LIN {X 0,Y 145.306,Z 169.772,A -85,B 0,C 180,E1 -24522.343,E2 -24522.343} C_VEL
LIN {X 0,Y 146.509,Z 171.03,A -85,B 0,C 180,E1 -24522.943,E2 -24522.943} C_VEL
LIN {X 0,Y 148.712,Z 174.406,A -85,B 0,C 180,E1 -24524.074,E2 -24524.074} C_VEL
LIN {X 0,Y 152.72,Z 180.292,A -85,B 0,C 180,E1 -24525.978,E2 -24525.978} C_VEL
LIN {X 0,Y 157.75,Z 189.892,A -85,B 0,C 180,E1 -24528.287,E2 -24528.287} C_VEL
LIN {X 0,Y 163.669,Z 203.505,A -85,B 0,C 180,E1 -24530.86,E2 -24530.86} C_VEL
LIN {X 0,Y 165.632,Z 209.272,A -85,B 0,C 180,E1 -24531.721,E2 -24531.721} C_VEL
LIN {X 0,Y 166.47,Z 218.611,A -85,B 0,C 180,E1 -24532.446,E2 -24532.446} C_VEL
LIN {X 0,Y 165.086,Z 241.604,A -85,B 0,C 180,E1 -24533.417,E2 -24533.417} C_VEL
LIN {X 0,Y 163.759,Z 252.442,A -85,B 0,C 180,E1 -24534.195,E2 -24534.195} C_VEL
LIN {X 0,Y 161.522,Z 264.21,A -85,B 0,C 180,E1 -24535.554,E2 -24535.554} C_VEL
LIN {X 0,Y 159.643,Z 271.971,A -85,B 0,C 180,E1 -24536.766,E2 -24536.766} C_VEL
LIN {X 0,Y 157.428,Z 279.918,A -85,B 0,C 180,E1 -24538.363,E2 -24538.363} C_VEL
LIN {X 0,Y 154.747,Z 287.967,A -85,B 0,C 180,E1 -24540.404,E2 -24540.404} C_VEL
LIN {X 0,Y 152.242,Z 294.615,A -85,B 0,C 180,E1 -24542.508,E2 -24542.508} C_VEL
LIN {X 0,Y 149.733,Z 300.93,A -85,B 0,C 180,E1 -24545.013,E2 -24545.013} C_VEL
LIN {X 0,Y 147.469,Z 306.176,A -85,B 0,C 180,E1 -24547.589,E2 -24547.589} C_VEL
LIN {X 0,Y 145.528,Z 310.551,A -85,B 0,C 180,E1 -24550.243,E2 -24550.243} C_VEL
LIN {X 0,Y 143.291,Z 315.716,A -85,B 0,C 180,E1 -24554.351,E2 -24554.351} C_VEL
LIN {X 0,Y 141.729,Z 319.509,A -85,B 0,C 180,E1 -24558.56,E2 -24558.56} C_VEL
LIN {X 0,Y 141.028,Z 321.248,A -85,B 0,C 180,E1 -24561.403,E2 -24561.403} C_VEL
LIN {X 0,Y 140.636,Z 322.494,A -85,B 0,C 180,E1 -24564.265,E2 -24564.265} C_VEL
LIN {X 0,Y 140.489,Z 323.267,A -85,B 0,C 180,E1 -24567.133,E2 -24567.133} C_VEL
LIN {X 0,Y 140.527,Z 323.559,A -85,B 0,C 180,E1 -24570.001,E2 -24570.001} C_VEL
LIN {X 0,Y 140.489,Z 323.255,A -85,B 0,C 180,E1 -24572.868,E2 -24572.868} C_VEL
LIN {X 0,Y 140.635,Z 322.459,A -85,B 0,C 180,E1 -24575.737,E2 -24575.737} C_VEL
LIN {X 0,Y 141.018,Z 321.189,A -85,B 0,C 180,E1 -24578.599,E2 -24578.599} C_VEL
LIN {X 0,Y 142.198,Z 318.101,A -85,B 0,C 180,E1 -24583.058,E2 -24583.058} C_VEL
LIN {X 0,Y 143.967,Z 314.085,A -85,B 0,C 180,E1 -24587.032,E2 -24587.032} C_VEL
LIN {X 0,Y 146.467,Z 308.354,A -85,B 0,C 180,E1 -24591.093,E2 -24591.093} C_VEL
LIN {X 0,Y 148.407,Z 303.949,A -85,B 0,C 180,E1 -24593.51,E2 -24593.51} C_VEL
LIN {X 0,Y 149.365,Z 300.401,A -85,B 0,C 180,E1 -24595.293,E2 -24595.293} C_VEL
LIN {X 0,Y 149.331,Z 294.144,A -85,B 0,C 180,E1 -24598.252,E2 -24598.252} C_VEL
LIN {X 0,Y 149.369,Z 287.186,A -85,B 0,C 180,E1 -24600.965,E2 -24600.965} C_VEL
LIN {X 0,Y 150.382,Z 282.536,A -85,B 0,C 180,E1 -24602.304,E2 -24602.304} C_VEL
LIN {X 0,Y 152.699,Z 275.158,A -85,B 0,C 180,E1 -24603.961,E2 -24603.961} C_VEL
LIN {X 0,Y 154.808,Z 267.286,A -85,B 0,C 180,E1 -24605.368,E2 -24605.368} C_VEL
LIN {X 0,Y 156.648,Z 258.957,A -85,B 0,C 180,E1 -24606.521,E2 -24606.521} C_VEL
LIN {X 0,Y 158.362,Z 249.266,A -85,B 0,C 180,E1 -24607.478,E2 -24607.478} C_VEL
LIN {X 0,Y 159.434,Z 239.95,A -85,B 0,C 180,E1 -24608.108,E2 -24608.108} C_VEL
LIN {X 0,Y 160.713,Z 217.708,A -85,B 0,C 180,E1 -24609.076,E2 -24609.076} C_VEL
LIN {X 0,Y 159.799,Z 210.505,A -85,B 0,C 180,E1 -24609.751,E2 -24609.751} C_VEL
LIN {X 0,Y 156.697,Z 202.354,A -85,B 0,C 180,E1 -24611.18,E2 -24611.18} C_VEL
LIN {X 0,Y 151.188,Z 189.975,A -85,B 0,C 180,E1 -24613.813,E2 -24613.813} C_VEL
LIN {X 0,Y 147.611,Z 183.574,A -85,B 0,C 180,E1 -24615.587,E2 -24615.587} C_VEL
LIN {X 0,Y 144.362,Z 178.907,A -85,B 0,C 180,E1 -24617.245,E2 -24617.245} C_VEL
LIN {X 0,Y 142.077,Z 175.537,A -85,B 0,C 180,E1 -24618.496,E2 -24618.496} C_VEL
LIN {X 0,Y 139.925,Z 172.519,A -85,B 0,C 180,E1 -24619.73,E2 -24619.73} C_VEL
LIN {X 0,Y 139.2,Z 171.415,A -85,B 0,C 180,E1 -24620.169,E2 -24620.169} C_VEL
LIN {X 0,Y 137.076,Z 169.279,A -85,B 0,C 180,E1 -24621.414,E2 -24621.414} C_VEL
LIN {X 0,Y 136.185,Z 167.112,A -85,B 0,C 180,E1 -24622.206,E2 -24622.206} C_VEL
LIN {X 0,Y 136.03,Z 166.393,A -85,B 0,C 180,E1 -24623.087,E2 -24623.087} C_VEL
LIN {X 0,Y 136.086,Z 166.344,A -85,B 0,C 180,E1 -24628.907,E2 -24628.907} C_VEL
LIN {X 0,Y 136.149,Z 166.308,A -85,B 0,C 180,E1 -24632.317,E2 -24632.317} C_VEL
LIN {X 0,Y 136.246,Z 166.297,A -85,B 0,C 180,E1 -24638.834,E2 -24638.834} C_VEL
LIN {X 0,Y 136.278,Z 166.322,A -85,B 0,C 180,E1 -24645.058,E2 -24645.058} C_VEL
LIN {X 0,Y 136.447,Z 166.265,A -85,B 0,C 180,E1 -24648.138,E2 -24648.138} C_VEL
LIN {X 0,Y 136.555,Z 166.253,A -85,B 0,C 180,E1 -24651.118,E2 -24651.118} C_VEL
LIN {X 0,Y 137.135,Z 166.174,A -85,B 0,C 180,E1 -24660,E2 -24660} C_VEL
LIN {X 0,Y 136.582,Z 166.243,A -85,B 0,C 180,E1 -24668.881,E2 -24668.881} C_VEL
LIN {X 0,Y 136.494,Z 166.277,A -85,B 0,C 180,E1 -24671.955,E2 -24671.955} C_VEL
LIN {X 0,Y 136.254,Z 166.287,A -85,B 0,C 180,E1 -24678.028,E2 -24678.028} C_VEL
LIN {X 0,Y 136.205,Z 166.325,A -85,B 0,C 180,E1 -24681.754,E2 -24681.754} C_VEL
LIN {X 0,Y 136.121,Z 166.321,A -85,B 0,C 180,E1 -24688.63,E2 -24688.63} C_VEL
LIN {X 0,Y 136.046,Z 166.327,A -85,B 0,C 180,E1 -24694.629,E2 -24694.629} C_VEL
LIN {X 0,Y 136.087,Z 166.637,A -85,B 0,C 180,E1 -24697.709,E2 -24697.709} C_VEL
LIN {X 0,Y 136.369,Z 167.781,A -85,B 0,C 180,E1 -24698.358,E2 -24698.358} C_VEL
LIN {X 0,Y 137.896,Z 170.333,A -85,B 0,C 180,E1 -24699.393,E2 -24699.393} C_VEL
LIN {X 0,Y 139.623,Z 171.907,A -85,B 0,C 180,E1 -24700.376,E2 -24700.376} C_VEL
LIN {X 0,Y 141.835,Z 175.359,A -85,B 0,C 180,E1 -24701.68,E2 -24701.68} C_VEL
LIN {X 0,Y 143.196,Z 177.113,A -85,B 0,C 180,E1 -24702.42,E2 -24702.42} C_VEL
LIN {X 0,Y 148.232,Z 184.462,A -85,B 0,C 180,E1 -24705.016,E2 -24705.016} C_VEL
LIN {X 0,Y 154.436,Z 194.858,A -85,B 0,C 180,E1 -24707.927,E2 -24707.927} C_VEL
LIN {X 0,Y 158.358,Z 202.506,A -85,B 0,C 180,E1 -24709.65,E2 -24709.65} C_VEL
LIN {X 0,Y 161.183,Z 209.91,A -85,B 0,C 180,E1 -24710.921,E2 -24710.921} C_VEL
LIN {X 0,Y 159.528,Z 236.911,A -85,B 0,C 180,E1 -24712.08,E2 -24712.08} C_VEL
LIN {X 0,Y 158.138,Z 248.435,A -85,B 0,C 180,E1 -24712.962,E2 -24712.962} C_VEL
LIN {X 0,Y 156.015,Z 259.714,A -85,B 0,C 180,E1 -24714.358,E2 -24714.358} C_VEL
LIN {X 0,Y 153.691,Z 269.059,A -85,B 0,C 180,E1 -24715.937,E2 -24715.937} C_VEL
LIN {X 0,Y 151.299,Z 277.142,A -85,B 0,C 180,E1 -24717.711,E2 -24717.711} C_VEL
LIN {X 0,Y 148.543,Z 284.842,A -85,B 0,C 180,E1 -24719.821,E2 -24719.821} C_VEL
LIN {X 0,Y 145.37,Z 292.896,A -85,B 0,C 180,E1 -24722.658,E2 -24722.658} C_VEL
LIN {X 0,Y 142.292,Z 299.943,A -85,B 0,C 180,E1 -24725.953,E2 -24725.953} C_VEL
LIN {X 0,Y 139.612,Z 305.513,A -85,B 0,C 180,E1 -24729.367,E2 -24729.367} C_VEL
LIN {X 0,Y 137.099,Z 310.686,A -85,B 0,C 180,E1 -24733.623,E2 -24733.623} C_VEL
LIN {X 0,Y 135.79,Z 313.338,A -85,B 0,C 180,E1 -24736.531,E2 -24736.531} C_VEL
LIN {X 0,Y 134.441,Z 316.24,A -85,B 0,C 180,E1 -24740.976,E2 -24740.976} C_VEL
LIN {X 0,Y 133.881,Z 317.504,A -85,B 0,C 180,E1 -24743.973,E2 -24743.973} C_VEL
LIN {X 0,Y 133.534,Z 318.299,A -85,B 0,C 180,E1 -24746.982,E2 -24746.982} C_VEL
LIN {X 0,Y 133.475,Z 318.601,A -85,B 0,C 180,E1 -24749.999,E2 -24749.999} C_VEL
LIN {X 0,Y 133.534,Z 318.32,A -85,B 0,C 180,E1 -24753.016,E2 -24753.016} C_VEL
LIN {X 0,Y 133.877,Z 317.568,A -85,B 0,C 180,E1 -24756.026,E2 -24756.026} C_VEL
LIN {X 0,Y 134.371,Z 316.349,A -85,B 0,C 180,E1 -24759.027,E2 -24759.027} C_VEL
LIN {X 0,Y 135.782,Z 313.49,A -85,B 0,C 180,E1 -24763.468,E2 -24763.468} C_VEL
LIN {X 0,Y 137.051,Z 310.887,A -85,B 0,C 180,E1 -24766.381,E2 -24766.381} C_VEL
LIN {X 0,Y 139.57,Z 305.767,A -85,B 0,C 180,E1 -24770.638,E2 -24770.638} C_VEL
LIN {X 0,Y 142.234,Z 300.257,A -85,B 0,C 180,E1 -24774.056,E2 -24774.056} C_VEL
LIN {X 0,Y 145.279,Z 293.329,A -85,B 0,C 180,E1 -24777.359,E2 -24777.359} C_VEL
LIN {X 0,Y 148.49,Z 285.371,A -85,B 0,C 180,E1 -24780.19,E2 -24780.19} C_VEL
LIN {X 0,Y 151.263,Z 277.782,A -85,B 0,C 180,E1 -24782.296,E2 -24782.296} C_VEL
LIN {X 0,Y 153.628,Z 269.829,A -85,B 0,C 180,E1 -24784.082,E2 -24784.082} C_VEL
LIN {X 0,Y 155.656,Z 262.251,A -85,B 0,C 180,E1 -24785.403,E2 -24785.403} C_VEL
LIN {X 0,Y 157.548,Z 252.986,A -85,B 0,C 180,E1 -24786.671,E2 -24786.671} C_VEL
LIN {X 0,Y 158.99,Z 243.674,A -85,B 0,C 180,E1 -24787.591,E2 -24787.591} C_VEL
LIN {X 0,Y 159.965,Z 233.274,A -85,B 0,C 180,E1 -24788.286,E2 -24788.286} C_VEL
LIN {X 0,Y 161.313,Z 209.971,A -85,B 0,C 180,E1 -24789.247,E2 -24789.247} C_VEL
LIN {X 0,Y 157.275,Z 199.981,A -85,B 0,C 180,E1 -24791.055,E2 -24791.055} C_VEL
LIN {X 0,Y 151.741,Z 190.114,A -85,B 0,C 180,E1 -24793.537,E2 -24793.537} C_VEL
LIN {X 0,Y 145.574,Z 180.386,A -85,B 0,C 180,E1 -24796.579,E2 -24796.579} C_VEL
LIN {X 0,Y 142.966,Z 176.681,A -85,B 0,C 180,E1 -24797.972,E2 -24797.972} C_VEL
LIN {X 0,Y 139.995,Z 172.674,A -85,B 0,C 180,E1 -24799.655,E2 -24799.655} C_VEL
LIN {X 0,Y 139.171,Z 171.41,A -85,B 0,C 180,E1 -24800.157,E2 -24800.157} C_VEL
LIN {X 0,Y 136.985,Z 169.121,A -85,B 0,C 180,E1 -24801.459,E2 -24801.459} C_VEL
LIN {X 0,Y 136.181,Z 167.095,A -85,B 0,C 180,E1 -24802.204,E2 -24802.204} C_VEL
LIN {X 0,Y 136.027,Z 166.389,A -85,B 0,C 180,E1 -24803.085,E2 -24803.085} C_VEL
LIN {X 0,Y 136.066,Z 166.34,A -85,B 0,C 180,E1 -24808.901,E2 -24808.901} C_VEL
LIN {X 0,Y 136.147,Z 166.311,A -85,B 0,C 180,E1 -24812.316,E2 -24812.316} C_VEL
LIN {X 0,Y 136.247,Z 166.312,A -85,B 0,C 180,E1 -24818.833,E2 -24818.833} C_VEL
LIN {X 0,Y 136.283,Z 166.31,A -85,B 0,C 180,E1 -24825.057,E2 -24825.057} C_VEL
LIN {X 0,Y 136.496,Z 166.277,A -85,B 0,C 180,E1 -24828.114,E2 -24828.114} C_VEL
LIN {X 0,Y 136.578,Z 166.243,A -85,B 0,C 180,E1 -24831.119,E2 -24831.119} C_VEL
LIN {X 0,Y 137.133,Z 166.175,A -85,B 0,C 180,E1 -24840,E2 -24840} C_VEL
LIN {X 0,Y 136.591,Z 166.249,A -85,B 0,C 180,E1 -24848.879,E2 -24848.879} C_VEL
LIN {X 0,Y 136.49,Z 166.261,A -85,B 0,C 180,E1 -24851.954,E2 -24851.954} C_VEL
LIN {X 0,Y 136.251,Z 166.296,A -85,B 0,C 180,E1 -24858.028,E2 -24858.028} C_VEL
LIN {X 0,Y 136.197,Z 166.309,A -85,B 0,C 180,E1 -24861.749,E2 -24861.749} C_VEL
LIN {X 0,Y 136.117,Z 166.314,A -85,B 0,C 180,E1 -24868.63,E2 -24868.63} C_VEL
LIN {X 0,Y 136.043,Z 166.328,A -85,B 0,C 180,E1 -24874.629,E2 -24874.629} C_VEL
LIN {X 0,Y 136.07,Z 166.645,A -85,B 0,C 180,E1 -24877.19,E2 -24877.19} C_VEL
LIN {X 0,Y 136.364,Z 167.734,A -85,B 0,C 180,E1 -24877.852,E2 -24877.852} C_VEL
LIN {X 0,Y 137.89,Z 170.334,A -85,B 0,C 180,E1 -24878.902,E2 -24878.902} C_VEL
LIN {X 0,Y 139.615,Z 171.833,A -85,B 0,C 180,E1 -24879.885,E2 -24879.885} C_VEL
LIN {X 0,Y 141.706,Z 175.185,A -85,B 0,C 180,E1 -24881.136,E2 -24881.136} C_VEL
LIN {X 0,Y 143.181,Z 177.043,A -85,B 0,C 180,E1 -24881.941,E2 -24881.941} C_VEL
LIN {X 0,Y 148.421,Z 184.735,A -85,B 0,C 180,E1 -24884.658,E2 -24884.658} C_VEL
LIN {X 0,Y 153.079,Z 193.843,A -85,B 0,C 180,E1 -24886.964,E2 -24886.964} C_VEL
LIN {X 0,Y 159.051,Z 207.999,A -85,B 0,C 180,E1 -24889.758,E2 -24889.758} C_VEL
LIN {X 0,Y 160.238,Z 211.76,A -85,B 0,C 180,E1 -24890.33,E2 -24890.33} C_VEL
LIN {X 0,Y 160.859,Z 219.504,A -85,B 0,C 180,E1 -24890.949,E2 -24890.949} C_VEL
LIN {X 0,Y 159.439,Z 241.491,A -85,B 0,C 180,E1 -24891.895,E2 -24891.895} C_VEL
LIN {X 0,Y 157.96,Z 253.007,A -85,B 0,C 180,E1 -24892.753,E2 -24892.753} C_VEL
LIN {X 0,Y 155.717,Z 264.088,A -85,B 0,C 180,E1 -24894.075,E2 -24894.075} C_VEL
LIN {X 0,Y 153.481,Z 272.848,A -85,B 0,C 180,E1 -24895.51,E2 -24895.51} C_VEL
LIN {X 0,Y 151.018,Z 281.024,A -85,B 0,C 180,E1 -24897.249,E2 -24897.249} C_VEL
LIN {X 0,Y 148.226,Z 288.863,A -85,B 0,C 180,E1 -24899.357,E2 -24899.357} C_VEL
LIN {X 0,Y 145.323,Z 296.197,A -85,B 0,C 180,E1 -24901.868,E2 -24901.868} C_VEL
LIN {X 0,Y 142.115,Z 303.636,A -85,B 0,C 180,E1 -24905.144,E2 -24905.144} C_VEL
LIN {X 0,Y 139.371,Z 309.466,A -85,B 0,C 180,E1 -24908.557,E2 -24908.557} C_VEL
LIN {X 0,Y 137.189,Z 314.066,A -85,B 0,C 180,E1 -24912.1,E2 -24912.1} C_VEL
LIN {X 0,Y 135.811,Z 317.057,A -85,B 0,C 180,E1 -24915.005,E2 -24915.005} C_VEL
LIN {X 0,Y 134.77,Z 319.381,A -85,B 0,C 180,E1 -24917.961,E2 -24917.961} C_VEL
LIN {X 0,Y 134.003,Z 321.12,A -85,B 0,C 180,E1 -24920.948,E2 -24920.948} C_VEL
LIN {X 0,Y 133.566,Z 322.365,A -85,B 0,C 180,E1 -24923.96,E2 -24923.96} C_VEL
LIN {X 0,Y 133.401,Z 323.138,A -85,B 0,C 180,E1 -24926.981,E2 -24926.981} C_VEL
LIN {X 0,Y 133.448,Z 323.431,A -85,B 0,C 180,E1 -24930.001,E2 -24930.001} C_VEL
LIN {X 0,Y 133.401,Z 323.126,A -85,B 0,C 180,E1 -24933.021,E2 -24933.021} C_VEL
LIN {X 0,Y 133.565,Z 322.33,A -85,B 0,C 180,E1 -24936.042,E2 -24936.042} C_VEL
LIN {X 0,Y 133.992,Z 321.06,A -85,B 0,C 180,E1 -24939.054,E2 -24939.054} C_VEL
LIN {X 0,Y 135.202,Z 318.139,A -85,B 0,C 180,E1 -24943.528,E2 -24943.528} C_VEL
LIN {X 0,Y 136.426,Z 315.477,A -85,B 0,C 180,E1 -24946.46,E2 -24946.46} C_VEL
LIN {X 0,Y 138.841,Z 310.281,A -85,B 0,C 180,E1 -24950.753,E2 -24950.753} C_VEL
LIN {X 0,Y 142.111,Z 303.43,A -85,B 0,C 180,E1 -24954.858,E2 -24954.858} C_VEL
LIN {X 0,Y 145.329,Z 295.948,A -85,B 0,C 180,E1 -24958.133,E2 -24958.133} C_VEL
LIN {X 0,Y 148.195,Z 288.568,A -85,B 0,C 180,E1 -24960.652,E2 -24960.652} C_VEL
LIN {X 0,Y 150.382,Z 282.536,A -85,B 0,C 180,E1 -24962.304,E2 -24962.304} C_VEL
LIN {X 0,Y 151.374,Z 277.866,A -85,B 0,C 180,E1 -24963.554,E2 -24963.554} C_VEL
LIN {X 0,Y 151.28,Z 269.925,A -85,B 0,C 180,E1 -24965.711,E2 -24965.711} C_VEL
LIN {X 0,Y 151.137,Z 261.247,A -85,B 0,C 180,E1 -24967.658,E2 -24967.658} C_VEL
LIN {X 0,Y 151.671,Z 255.69,A -85,B 0,C 180,E1 -24968.473,E2 -24968.473} C_VEL
LIN {X 0,Y 153.583,Z 243.837,A -85,B 0,C 180,E1 -24969.505,E2 -24969.505} C_VEL
LIN {X 0,Y 154.8,Z 226.982,A -85,B 0,C 180,E1 -24970.312,E2 -24970.312} C_VEL
LIN {X 0,Y 155.171,Z 218.327,A -85,B 0,C 180,E1 -24970.711,E2 -24970.711} C_VEL
LIN {X 0,Y 154.459,Z 212.838,A -85,B 0,C 180,E1 -24971.269,E2 -24971.269} C_VEL
LIN {X 0,Y 149.342,Z 199.941,A -85,B 0,C 180,E1 -24973.84,E2 -24973.84} C_VEL
LIN {X 0,Y 144.771,Z 190.32,A -85,B 0,C 180,E1 -24976.265,E2 -24976.265} C_VEL
LIN {X 0,Y 140.402,Z 183.75,A -85,B 0,C 180,E1 -24978.646,E2 -24978.646} C_VEL
LIN {X 0,Y 138.218,Z 180.588,A -85,B 0,C 180,E1 -24979.928,E2 -24979.928} C_VEL
LIN {X 0,Y 135.858,Z 177.165,A -85,B 0,C 180,E1 -24981.402,E2 -24981.402} C_VEL
LIN {X 0,Y 133.57,Z 174.376,A -85,B 0,C 180,E1 -24982.883,E2 -24982.883} C_VEL
LIN {X 0,Y 132.566,Z 172.525,A -85,B 0,C 180,E1 -24983.623,E2 -24983.623} C_VEL
LIN {X 0,Y 130.346,Z 170.554,A -85,B 0,C 180,E1 -24985.146,E2 -24985.146} C_VEL
LIN {X 0,Y 129.15,Z 167.989,A -85,B 0,C 180,E1 -24986.323,E2 -24986.323} C_VEL
LIN {X 0,Y 129.005,Z 167.269,A -85,B 0,C 180,E1 -24987.455,E2 -24987.455} C_VEL
LIN {X 0,Y 129.052,Z 167.197,A -85,B 0,C 180,E1 -24990.652,E2 -24990.652} C_VEL
LIN {X 0,Y 129.109,Z 167.195,A -85,B 0,C 180,E1 -24997.728,E2 -24997.728} C_VEL
LIN {X 0,Y 129.159,Z 167.173,A -85,B 0,C 180,E1 -25000.945,E2 -25000.945} C_VEL
LIN {X 0,Y 129.369,Z 167.147,A -85,B 0,C 180,E1 -25007.922,E2 -25007.922} C_VEL
LIN {X 0,Y 129.48,Z 167.13,A -85,B 0,C 180,E1 -25010.629,E2 -25010.629} C_VEL
LIN {X 0,Y 129.675,Z 167.113,A -85,B 0,C 180,E1 -25016.894,E2 -25016.894} C_VEL
LIN {X 0,Y 130.09,Z 167.05,A -85,B 0,C 180,E1 -25020,E2 -25020} C_VEL
LIN {X 0,Y 129.51,Z 167.123,A -85,B 0,C 180,E1 -25029.37,E2 -25029.37} C_VEL
LIN {X 0,Y 129.396,Z 167.168,A -85,B 0,C 180,E1 -25032.548,E2 -25032.548} C_VEL
LIN {X 0,Y 129.163,Z 167.171,A -85,B 0,C 180,E1 -25039.055,E2 -25039.055} C_VEL
LIN {X 0,Y 129.112,Z 167.214,A -85,B 0,C 180,E1 -25042.398,E2 -25042.398} C_VEL
LIN {X 0,Y 129.053,Z 167.208,A -85,B 0,C 180,E1 -25049.349,E2 -25049.349} C_VEL
LIN {X 0,Y 129.016,Z 167.477,A -85,B 0,C 180,E1 -25053.48,E2 -25053.48} C_VEL
LIN {X 0,Y 129.294,Z 168.453,A -85,B 0,C 180,E1 -25054.229,E2 -25054.229} C_VEL
LIN {X 0,Y 130.744,Z 171.071,A -85,B 0,C 180,E1 -25055.45,E2 -25055.45} C_VEL
LIN {X 0,Y 132.851,Z 172.914,A -85,B 0,C 180,E1 -25056.877,E2 -25056.877} C_VEL
LIN {X 0,Y 134.81,Z 176.099,A -85,B 0,C 180,E1 -25058.249,E2 -25058.249} C_VEL
LIN {X 0,Y 136.534,Z 178.074,A -85,B 0,C 180,E1 -25059.324,E2 -25059.324} C_VEL
LIN {X 0,Y 139.008,Z 181.522,A -85,B 0,C 180,E1 -25060.828,E2 -25060.828} C_VEL
LIN {X 0,Y 144.882,Z 190.467,A -85,B 0,C 180,E1 -25064.091,E2 -25064.091} C_VEL
LIN {X 0,Y 149.951,Z 199.143,A -85,B 0,C 180,E1 -25066.63,E2 -25066.63} C_VEL
LIN {X 0,Y 153.651,Z 206.532,A -85,B 0,C 180,E1 -25068.381,E2 -25068.381} C_VEL
LIN {X 0,Y 155.653,Z 211.817,A -85,B 0,C 180,E1 -25069.352,E2 -25069.352} C_VEL
LIN {X 0,Y 153.999,Z 237.056,A -85,B 0,C 180,E1 -25070.459,E2 -25070.459} C_VEL
LIN {X 0,Y 152.596,Z 248.166,A -85,B 0,C 180,E1 -25071.317,E2 -25071.317} C_VEL
LIN {X 0,Y 150.548,Z 258.884,A -85,B 0,C 180,E1 -25072.635,E2 -25072.635} C_VEL
LIN {X 0,Y 148.259,Z 267.964,A -85,B 0,C 180,E1 -25074.163,E2 -25074.163} C_VEL
LIN {X 0,Y 145.762,Z 276.046,A -85,B 0,C 180,E1 -25075.908,E2 -25075.908} C_VEL
LIN {X 0,Y 142.874,Z 283.954,A -85,B 0,C 180,E1 -25078.075,E2 -25078.075} C_VEL
LIN {X 0,Y 139.844,Z 291.329,A -85,B 0,C 180,E1 -25080.659,E2 -25080.659} C_VEL
LIN {X 0,Y 136.435,Z 298.8,A -85,B 0,C 180,E1 -25084.033,E2 -25084.033} C_VEL
LIN {X 0,Y 133,Z 305.642,A -85,B 0,C 180,E1 -25088.29,E2 -25088.29} C_VEL
LIN {X 0,Y 130.308,Z 310.816,A -85,B 0,C 180,E1 -25092.744,E2 -25092.744} C_VEL
LIN {X 0,Y 128.901,Z 313.467,A -85,B 0,C 180,E1 -25095.797,E2 -25095.797} C_VEL
LIN {X 0,Y 127.429,Z 316.369,A -85,B 0,C 180,E1 -25100.475,E2 -25100.475} C_VEL
LIN {X 0,Y 126.83,Z 317.632,A -85,B 0,C 180,E1 -25103.636,E2 -25103.636} C_VEL
LIN {X 0,Y 126.458,Z 318.427,A -85,B 0,C 180,E1 -25106.813,E2 -25106.813} C_VEL
LIN {X 0,Y 126.391,Z 318.729,A -85,B 0,C 180,E1 -25109.999,E2 -25109.999} C_VEL
LIN {X 0,Y 126.458,Z 318.449,A -85,B 0,C 180,E1 -25113.185,E2 -25113.185} C_VEL
LIN {X 0,Y 126.824,Z 317.696,A -85,B 0,C 180,E1 -25116.362,E2 -25116.362} C_VEL
LIN {X 0,Y 127.377,Z 316.477,A -85,B 0,C 180,E1 -25119.527,E2 -25119.527} C_VEL
LIN {X 0,Y 128.892,Z 313.618,A -85,B 0,C 180,E1 -25124.203,E2 -25124.203} C_VEL
LIN {X 0,Y 130.265,Z 311.014,A -85,B 0,C 180,E1 -25127.261,E2 -25127.261} C_VEL
LIN {X 0,Y 132.961,Z 305.894,A -85,B 0,C 180,E1 -25131.715,E2 -25131.715} C_VEL
LIN {X 0,Y 135.782,Z 300.384,A -85,B 0,C 180,E1 -25135.277,E2 -25135.277} C_VEL
LIN {X 0,Y 139.021,Z 293.454,A -85,B 0,C 180,E1 -25138.701,E2 -25138.701} C_VEL
LIN {X 0,Y 142.41,Z 285.496,A -85,B 0,C 180,E1 -25141.623,E2 -25141.623} C_VEL
LIN {X 0,Y 145.329,Z 277.906,A -85,B 0,C 180,E1 -25143.788,E2 -25143.788} C_VEL
LIN {X 0,Y 147.738,Z 270.209,A -85,B 0,C 180,E1 -25145.57,E2 -25145.57} C_VEL
LIN {X 0,Y 150.21,Z 261.147,A -85,B 0,C 180,E1 -25147.169,E2 -25147.169} C_VEL
LIN {X 0,Y 151.988,Z 252.703,A -85,B 0,C 180,E1 -25148.318,E2 -25148.318} C_VEL
LIN {X 0,Y 153.494,Z 243.294,A -85,B 0,C 180,E1 -25149.251,E2 -25149.251} C_VEL
LIN {X 0,Y 154.558,Z 232.452,A -85,B 0,C 180,E1 -25149.962,E2 -25149.962} C_VEL
LIN {X 0,Y 155.753,Z 211.844,A -85,B 0,C 180,E1 -25150.833,E2 -25150.833} C_VEL
LIN {X 0,Y 152.399,Z 203.592,A -85,B 0,C 180,E1 -25152.451,E2 -25152.451} C_VEL
LIN {X 0,Y 147.336,Z 194.468,A -85,B 0,C 180,E1 -25154.898,E2 -25154.898} C_VEL
LIN {X 0,Y 141.743,Z 185.533,A -85,B 0,C 180,E1 -25157.865,E2 -25157.865} C_VEL
LIN {X 0,Y 138.218,Z 180.603,A -85,B 0,C 180,E1 -25159.901,E2 -25159.901} C_VEL
LIN {X 0,Y 135.769,Z 177.083,A -85,B 0,C 180,E1 -25161.442,E2 -25161.442} C_VEL
LIN {X 0,Y 133.459,Z 174.155,A -85,B 0,C 180,E1 -25162.965,E2 -25162.965} C_VEL
LIN {X 0,Y 132.572,Z 172.528,A -85,B 0,C 180,E1 -25163.624,E2 -25163.624} C_VEL
LIN {X 0,Y 130.362,Z 170.599,A -85,B 0,C 180,E1 -25165.151,E2 -25165.151} C_VEL
LIN {X 0,Y 129.075,Z 167.758,A -85,B 0,C 180,E1 -25166.537,E2 -25166.537} C_VEL
LIN {X 0,Y 128.976,Z 167.233,A -85,B 0,C 180,E1 -25167.908,E2 -25167.908} C_VEL
LIN {X 0,Y 129.05,Z 167.211,A -85,B 0,C 180,E1 -25170.65,E2 -25170.65} C_VEL
LIN {X 0,Y 129.109,Z 167.214,A -85,B 0,C 180,E1 -25177.724,E2 -25177.724} C_VEL
LIN {X 0,Y 129.16,Z 167.172,A -85,B 0,C 180,E1 -25180.944,E2 -25180.944} C_VEL
LIN {X 0,Y 129.415,Z 167.161,A -85,B 0,C 180,E1 -25187.821,E2 -25187.821} C_VEL
LIN {X 0,Y 129.507,Z 167.124,A -85,B 0,C 180,E1 -25190.63,E2 -25190.63} C_VEL
LIN {X 0,Y 130.089,Z 167.051,A -85,B 0,C 180,E1 -25200,E2 -25200} C_VEL
LIN {X 0,Y 129.516,Z 167.125,A -85,B 0,C 180,E1 -25209.369,E2 -25209.369} C_VEL
LIN {X 0,Y 129.393,Z 167.149,A -85,B 0,C 180,E1 -25212.548,E2 -25212.548} C_VEL
LIN {X 0,Y 129.158,Z 167.173,A -85,B 0,C 180,E1 -25219.055,E2 -25219.055} C_VEL
LIN {X 0,Y 129.107,Z 167.198,A -85,B 0,C 180,E1 -25222.398,E2 -25222.398} C_VEL
LIN {X 0,Y 129.058,Z 167.198,A -85,B 0,C 180,E1 -25229.392,E2 -25229.392} C_VEL
LIN {X 0,Y 129.018,Z 167.505,A -85,B 0,C 180,E1 -25232.948,E2 -25232.948} C_VEL
LIN {X 0,Y 129.324,Z 168.644,A -85,B 0,C 180,E1 -25233.744,E2 -25233.744} C_VEL
LIN {X 0,Y 131.007,Z 171.356,A -85,B 0,C 180,E1 -25235.115,E2 -25235.115} C_VEL
LIN {X 0,Y 132.887,Z 172.994,A -85,B 0,C 180,E1 -25236.393,E2 -25236.393} C_VEL
LIN {X 0,Y 134.957,Z 176.273,A -85,B 0,C 180,E1 -25237.844,E2 -25237.844} C_VEL
LIN {X 0,Y 136.565,Z 178.084,A -85,B 0,C 180,E1 -25238.849,E2 -25238.849} C_VEL
LIN {X 0,Y 140.484,Z 183.847,A -85,B 0,C 180,E1 -25241.225,E2 -25241.225} C_VEL
LIN {X 0,Y 144.593,Z 189.956,A -85,B 0,C 180,E1 -25243.477,E2 -25243.477} C_VEL
LIN {X 0,Y 148.776,Z 198.456,A -85,B 0,C 180,E1 -25245.708,E2 -25245.708} C_VEL
LIN {X 0,Y 154.408,Z 212.378,A -85,B 0,C 180,E1 -25248.556,E2 -25248.556} C_VEL
LIN {X 0,Y 155.035,Z 215.012,A -85,B 0,C 180,E1 -25248.918,E2 -25248.918} C_VEL
LIN {X 0,Y 155.386,Z 220.154,A -85,B 0,C 180,E1 -25249.337,E2 -25249.337} C_VEL
LIN {X 0,Y 153.922,Z 241.379,A -85,B 0,C 180,E1 -25250.266,E2 -25250.266} C_VEL
LIN {X 0,Y 152.484,Z 252.32,A -85,B 0,C 180,E1 -25251.091,E2 -25251.091} C_VEL
LIN {X 0,Y 150.033,Z 263.965,A -85,B 0,C 180,E1 -25252.487,E2 -25252.487} C_VEL
LIN {X 0,Y 147.554,Z 273.182,A -85,B 0,C 180,E1 -25254.042,E2 -25254.042} C_VEL
LIN {X 0,Y 145.103,Z 280.9,A -85,B 0,C 180,E1 -25255.734,E2 -25255.734} C_VEL
LIN {X 0,Y 142.174,Z 288.738,A -85,B 0,C 180,E1 -25257.901,E2 -25257.901} C_VEL
LIN {X 0,Y 139.084,Z 296.07,A -85,B 0,C 180,E1 -25260.484,E2 -25260.484} C_VEL
LIN {X 0,Y 135.676,Z 303.509,A -85,B 0,C 180,E1 -25263.878,E2 -25263.878} C_VEL
LIN {X 0,Y 132.788,Z 309.339,A -85,B 0,C 180,E1 -25267.437,E2 -25267.437} C_VEL
LIN {X 0,Y 130.44,Z 313.939,A -85,B 0,C 180,E1 -25271.14,E2 -25271.14} C_VEL
LIN {X 0,Y 128.952,Z 316.93,A -85,B 0,C 180,E1 -25274.188,E2 -25274.188} C_VEL
LIN {X 0,Y 127.838,Z 319.253,A -85,B 0,C 180,E1 -25277.298,E2 -25277.298} C_VEL
LIN {X 0,Y 126.982,Z 320.992,A -85,B 0,C 180,E1 -25280.443,E2 -25280.443} C_VEL
LIN {X 0,Y 126.491,Z 322.237,A -85,B 0,C 180,E1 -25283.621,E2 -25283.621} C_VEL
LIN {X 0,Y 126.309,Z 323.01,A -85,B 0,C 180,E1 -25286.811,E2 -25286.811} C_VEL
LIN {X 0,Y 126.359,Z 323.303,A -85,B 0,C 180,E1 -25290.001,E2 -25290.001} C_VEL
LIN {X 0,Y 126.309,Z 322.998,A -85,B 0,C 180,E1 -25293.19,E2 -25293.19} C_VEL
LIN {X 0,Y 126.49,Z 322.201,A -85,B 0,C 180,E1 -25296.381,E2 -25296.381} C_VEL
LIN {X 0,Y 126.971,Z 320.931,A -85,B 0,C 180,E1 -25299.559,E2 -25299.559} C_VEL
LIN {X 0,Y 128.286,Z 318.009,A -85,B 0,C 180,E1 -25304.273,E2 -25304.273} C_VEL
LIN {X 0,Y 129.612,Z 315.347,A -85,B 0,C 180,E1 -25307.352,E2 -25307.352} C_VEL
LIN {X 0,Y 132.212,Z 310.151,A -85,B 0,C 180,E1 -25311.846,E2 -25311.846} C_VEL
LIN {X 0,Y 135.673,Z 303.299,A -85,B 0,C 180,E1 -25316.124,E2 -25316.124} C_VEL
LIN {X 0,Y 139.099,Z 295.817,A -85,B 0,C 180,E1 -25319.514,E2 -25319.514} C_VEL
LIN {X 0,Y 142.144,Z 288.437,A -85,B 0,C 180,E1 -25322.108,E2 -25322.108} C_VEL
LIN {X 0,Y 145.055,Z 280.625,A -85,B 0,C 180,E1 -25324.249,E2 -25324.249} C_VEL
LIN {X 0,Y 147.764,Z 272.025,A -85,B 0,C 180,E1 -25326.098,E2 -25326.098} C_VEL
LIN {X 0,Y 150.379,Z 261.868,A -85,B 0,C 180,E1 -25327.753,E2 -25327.753} C_VEL
LIN {X 0,Y 151.671,Z 255.69,A -85,B 0,C 180,E1 -25328.473,E2 -25328.473} C_VEL
LIN {X 0,Y 152.155,Z 250.118,A -85,B 0,C 180,E1 -25329.187,E2 -25329.187} C_VEL
LIN {X 0,Y 151.719,Z 244.592,A -85,B 0,C 180,E1 -25330.004,E2 -25330.004} C_VEL
LIN {X 0,Y 149.645,Z 231.584,A -85,B 0,C 180,E1 -25331.715,E2 -25331.715} C_VEL
LIN {X 0,Y 149.529,Z 225.756,A -85,B 0,C 180,E1 -25332.117,E2 -25332.117} C_VEL
LIN {X 0,Y 149.795,Z 219.352,A -85,B 0,C 180,E1 -25332.43,E2 -25332.43} C_VEL
LIN {X 0,Y 149.289,Z 215.45,A -85,B 0,C 180,E1 -25332.857,E2 -25332.857} C_VEL
LIN {X 0,Y 144.343,Z 202.799,A -85,B 0,C 180,E1 -25335.568,E2 -25335.568} C_VEL
LIN {X 0,Y 140.337,Z 194.347,A -85,B 0,C 180,E1 -25337.88,E2 -25337.88} C_VEL
LIN {X 0,Y 135.001,Z 186.261,A -85,B 0,C 180,E1 -25341.099,E2 -25341.099} C_VEL
LIN {X 0,Y 132.454,Z 182.649,A -85,B 0,C 180,E1 -25342.792,E2 -25342.792} C_VEL
LIN {X 0,Y 129.985,Z 179.136,A -85,B 0,C 180,E1 -25344.568,E2 -25344.568} C_VEL
LIN {X 0,Y 126.977,Z 175.579,A -85,B 0,C 180,E1 -25346.869,E2 -25346.869} C_VEL
LIN {X 0,Y 125.983,Z 173.681,A -85,B 0,C 180,E1 -25347.762,E2 -25347.762} C_VEL
LIN {X 0,Y 123.38,Z 171.482,A -85,B 0,C 180,E1 -25349.969,E2 -25349.969} C_VEL
LIN {X 0,Y 122.072,Z 168.7,A -85,B 0,C 180,E1 -25351.655,E2 -25351.655} C_VEL
LIN {X 0,Y 121.944,Z 168.109,A -85,B 0,C 180,E1 -25353.009,E2 -25353.009} C_VEL
LIN {X 0,Y 122.026,Z 168.083,A -85,B 0,C 180,E1 -25357.149,E2 -25357.149} C_VEL
LIN {X 0,Y 122.116,Z 168.067,A -85,B 0,C 180,E1 -25363.276,E2 -25363.276} C_VEL
LIN {X 0,Y 122.32,Z 168.026,A -85,B 0,C 180,E1 -25367.624,E2 -25367.624} C_VEL
LIN {X 0,Y 122.43,Z 168.039,A -85,B 0,C 180,E1 -25373.408,E2 -25373.408} C_VEL
LIN {X 0,Y 123.044,Z 167.927,A -85,B 0,C 180,E1 -25380,E2 -25380} C_VEL
LIN {X 0,Y 122.416,Z 168.013,A -85,B 0,C 180,E1 -25387.092,E2 -25387.092} C_VEL
LIN {X 0,Y 122.365,Z 168.04,A -85,B 0,C 180,E1 -25392.472,E2 -25392.472} C_VEL
LIN {X 0,Y 122.12,Z 168.051,A -85,B 0,C 180,E1 -25396.724,E2 -25396.724} C_VEL
LIN {X 0,Y 122.028,Z 168.095,A -85,B 0,C 180,E1 -25402.853,E2 -25402.853} C_VEL
LIN {X 0,Y 122.003,Z 168.369,A -85,B 0,C 180,E1 -25408.202,E2 -25408.202} C_VEL
LIN {X 0,Y 122.379,Z 169.586,A -85,B 0,C 180,E1 -25409.254,E2 -25409.254} C_VEL
LIN {X 0,Y 123.802,Z 172.016,A -85,B 0,C 180,E1 -25410.725,E2 -25410.725} C_VEL
LIN {X 0,Y 126.234,Z 174.076,A -85,B 0,C 180,E1 -25412.758,E2 -25412.758} C_VEL
LIN {X 0,Y 128.108,Z 177.169,A -85,B 0,C 180,E1 -25414.349,E2 -25414.349} C_VEL
LIN {X 0,Y 129.957,Z 179.107,A -85,B 0,C 180,E1 -25415.712,E2 -25415.712} C_VEL
LIN {X 0,Y 132.432,Z 182.61,A -85,B 0,C 180,E1 -25417.491,E2 -25417.491} C_VEL
LIN {X 0,Y 138.312,Z 191.064,A -85,B 0,C 180,E1 -25421.235,E2 -25421.235} C_VEL
LIN {X 0,Y 144.54,Z 201.576,A -85,B 0,C 180,E1 -25424.726,E2 -25424.726} C_VEL
LIN {X 0,Y 148.69,Z 209.771,A -85,B 0,C 180,E1 -25426.861,E2 -25426.861} C_VEL
LIN {X 0,Y 150.172,Z 213.707,A -85,B 0,C 180,E1 -25427.642,E2 -25427.642} C_VEL
LIN {X 0,Y 148.609,Z 237.201,A -85,B 0,C 180,E1 -25428.722,E2 -25428.722} C_VEL
LIN {X 0,Y 147.003,Z 249.064,A -85,B 0,C 180,E1 -25429.668,E2 -25429.668} C_VEL
LIN {X 0,Y 144.972,Z 259.018,A -85,B 0,C 180,E1 -25430.933,E2 -25430.933} C_VEL
LIN {X 0,Y 142.492,Z 268.369,A -85,B 0,C 180,E1 -25432.55,E2 -25432.55} C_VEL
LIN {X 0,Y 139.942,Z 276.178,A -85,B 0,C 180,E1 -25434.28,E2 -25434.28} C_VEL
LIN {X 0,Y 136.916,Z 284.086,A -85,B 0,C 180,E1 -25436.508,E2 -25436.508} C_VEL
LIN {X 0,Y 133.713,Z 291.46,A -85,B 0,C 180,E1 -25439.171,E2 -25439.171} C_VEL
LIN {X 0,Y 130.09,Z 298.931,A -85,B 0,C 180,E1 -25442.663,E2 -25442.663} C_VEL
LIN {X 0,Y 126.445,Z 305.772,A -85,B 0,C 180,E1 -25447.103,E2 -25447.103} C_VEL
LIN {X 0,Y 123.558,Z 310.945,A -85,B 0,C 180,E1 -25451.769,E2 -25451.769} C_VEL
LIN {X 0,Y 122.019,Z 313.597,A -85,B 0,C 180,E1 -25454.977,E2 -25454.977} C_VEL
LIN {X 0,Y 120.445,Z 316.498,A -85,B 0,C 180,E1 -25459.918,E2 -25459.918} C_VEL
LIN {X 0,Y 119.775,Z 317.761,A -85,B 0,C 180,E1 -25463.26,E2 -25463.26} C_VEL
LIN {X 0,Y 119.375,Z 318.556,A -85,B 0,C 180,E1 -25466.624,E2 -25466.624} C_VEL
LIN {X 0,Y 119.294,Z 318.858,A -85,B 0,C 180,E1 -25469.999,E2 -25469.999} C_VEL
LIN {X 0,Y 119.375,Z 318.577,A -85,B 0,C 180,E1 -25473.374,E2 -25473.374} C_VEL
LIN {X 0,Y 119.768,Z 317.824,A -85,B 0,C 180,E1 -25476.739,E2 -25476.739} C_VEL
LIN {X 0,Y 120.372,Z 316.604,A -85,B 0,C 180,E1 -25480.087,E2 -25480.087} C_VEL
LIN {X 0,Y 122.009,Z 313.745,A -85,B 0,C 180,E1 -25485.022,E2 -25485.022} C_VEL
LIN {X 0,Y 123.501,Z 311.141,A -85,B 0,C 180,E1 -25488.238,E2 -25488.238} C_VEL
LIN {X 0,Y 126.389,Z 306.021,A -85,B 0,C 180,E1 -25492.906,E2 -25492.906} C_VEL
LIN {X 0,Y 129.378,Z 300.511,A -85,B 0,C 180,E1 -25496.624,E2 -25496.624} C_VEL
LIN {X 0,Y 132.851,Z 293.58,A -85,B 0,C 180,E1 -25500.169,E2 -25500.169} C_VEL
LIN {X 0,Y 136.427,Z 285.621,A -85,B 0,C 180,E1 -25503.184,E2 -25503.184} C_VEL
LIN {X 0,Y 139.5,Z 278.03,A -85,B 0,C 180,E1 -25505.405,E2 -25505.405} C_VEL
LIN {X 0,Y 141.985,Z 270.5,A -85,B 0,C 180,E1 -25507.198,E2 -25507.198} C_VEL
LIN {X 0,Y 144.414,Z 262.106,A -85,B 0,C 180,E1 -25508.733,E2 -25508.733} C_VEL
LIN {X 0,Y 146.457,Z 252.963,A -85,B 0,C 180,E1 -25510.023,E2 -25510.023} C_VEL
LIN {X 0,Y 148.054,Z 243.5,A -85,B 0,C 180,E1 -25510.981,E2 -25510.981} C_VEL
LIN {X 0,Y 149.192,Z 232.574,A -85,B 0,C 180,E1 -25511.71,E2 -25511.71} C_VEL
LIN {X 0,Y 150.39,Z 214.062,A -85,B 0,C 180,E1 -25512.489,E2 -25512.489} C_VEL
LIN {X 0,Y 147.746,Z 207.585,A -85,B 0,C 180,E1 -25513.866,E2 -25513.866} C_VEL
LIN {X 0,Y 143.029,Z 198.815,A -85,B 0,C 180,E1 -25516.34,E2 -25516.34} C_VEL
LIN {X 0,Y 137.982,Z 190.62,A -85,B 0,C 180,E1 -25519.228,E2 -25519.228} C_VEL
LIN {X 0,Y 134.74,Z 185.94,A -85,B 0,C 180,E1 -25521.25,E2 -25521.25} C_VEL
LIN {X 0,Y 132.519,Z 182.71,A -85,B 0,C 180,E1 -25522.75,E2 -25522.75} C_VEL
LIN {X 0,Y 129.95,Z 179.033,A -85,B 0,C 180,E1 -25524.615,E2 -25524.615} C_VEL
LIN {X 0,Y 127.015,Z 175.607,A -85,B 0,C 180,E1 -25526.879,E2 -25526.879} C_VEL
LIN {X 0,Y 126.031,Z 173.684,A -85,B 0,C 180,E1 -25527.775,E2 -25527.775} C_VEL
LIN {X 0,Y 123.429,Z 171.57,A -85,B 0,C 180,E1 -25529.995,E2 -25529.995} C_VEL
LIN {X 0,Y 122.055,Z 168.675,A -85,B 0,C 180,E1 -25531.811,E2 -25531.811} C_VEL
LIN {X 0,Y 121.964,Z 168.097,A -85,B 0,C 180,E1 -25533.475,E2 -25533.475} C_VEL
LIN {X 0,Y 122.049,Z 168.065,A -85,B 0,C 180,E1 -25539.787,E2 -25539.787} C_VEL
LIN {X 0,Y 122.284,Z 168.064,A -85,B 0,C 180,E1 -25546.709,E2 -25546.709} C_VEL
LIN {X 0,Y 122.439,Z 168.005,A -85,B 0,C 180,E1 -25550.084,E2 -25550.084} C_VEL
LIN {X 0,Y 122.605,Z 168.019,A -85,B 0,C 180,E1 -25556.714,E2 -25556.714} C_VEL
LIN {X 0,Y 123.043,Z 167.927,A -85,B 0,C 180,E1 -25560,E2 -25560} C_VEL
LIN {X 0,Y 122.448,Z 168.036,A -85,B 0,C 180,E1 -25566.591,E2 -25566.591} C_VEL
LIN {X 0,Y 122.445,Z 168.003,A -85,B 0,C 180,E1 -25569.915,E2 -25569.915} C_VEL
LIN {X 0,Y 122.263,Z 168.044,A -85,B 0,C 180,E1 -25573.293,E2 -25573.293} C_VEL
LIN {X 0,Y 122.047,Z 168.058,A -85,B 0,C 180,E1 -25580.212,E2 -25580.212} C_VEL
LIN {X 0,Y 121.962,Z 168.112,A -85,B 0,C 180,E1 -25586.525,E2 -25586.525} C_VEL
LIN {X 0,Y 122.073,Z 168.705,A -85,B 0,C 180,E1 -25588.037,E2 -25588.037} C_VEL
LIN {X 0,Y 123.614,Z 171.779,A -85,B 0,C 180,E1 -25589.969,E2 -25589.969} C_VEL
LIN {X 0,Y 126.205,Z 174.01,A -85,B 0,C 180,E1 -25592.175,E2 -25592.175} C_VEL
LIN {X 0,Y 128.274,Z 177.348,A -85,B 0,C 180,E1 -25593.938,E2 -25593.938} C_VEL
LIN {X 0,Y 129.98,Z 179.095,A -85,B 0,C 180,E1 -25595.2,E2 -25595.2} C_VEL
LIN {X 0,Y 132.507,Z 182.7,A -85,B 0,C 180,E1 -25597.033,E2 -25597.033} C_VEL
LIN {X 0,Y 133.779,Z 184.443,A -85,B 0,C 180,E1 -25597.895,E2 -25597.895} C_VEL
LIN {X 0,Y 138.712,Z 191.715,A -85,B 0,C 180,E1 -25600.996,E2 -25600.996} C_VEL
LIN {X 0,Y 141.717,Z 196.898,A -85,B 0,C 180,E1 -25602.75,E2 -25602.75} C_VEL
LIN {X 0,Y 146.302,Z 207.357,A -85,B 0,C 180,E1 -25605.361,E2 -25605.361} C_VEL
LIN {X 0,Y 149.716,Z 216.415,A -85,B 0,C 180,E1 -25607.215,E2 -25607.215} C_VEL
LIN {X 0,Y 149.981,Z 221.378,A -85,B 0,C 180,E1 -25607.624,E2 -25607.624} C_VEL
LIN {X 0,Y 148.529,Z 241.267,A -85,B 0,C 180,E1 -25608.515,E2 -25608.515} C_VEL
LIN {X 0,Y 147.071,Z 252.018,A -85,B 0,C 180,E1 -25609.342,E2 -25609.342} C_VEL
LIN {X 0,Y 144.867,Z 262.353,A -85,B 0,C 180,E1 -25610.544,E2 -25610.544} C_VEL
LIN {X 0,Y 142.031,Z 272.504,A -85,B 0,C 180,E1 -25612.244,E2 -25612.244} C_VEL
LIN {X 0,Y 139.23,Z 280.957,A -85,B 0,C 180,E1 -25614.137,E2 -25614.137} C_VEL
LIN {X 0,Y 136.224,Z 288.613,A -85,B 0,C 180,E1 -25616.317,E2 -25616.317} C_VEL
LIN {X 0,Y 132.926,Z 295.944,A -85,B 0,C 180,E1 -25618.97,E2 -25618.97} C_VEL
LIN {X 0,Y 129.327,Z 303.383,A -85,B 0,C 180,E1 -25622.49,E2 -25622.49} C_VEL
LIN {X 0,Y 126.226,Z 309.212,A -85,B 0,C 180,E1 -25626.193,E2 -25626.193} C_VEL
LIN {X 0,Y 123.715,Z 313.811,A -85,B 0,C 180,E1 -25630.072,E2 -25630.072} C_VEL
LIN {X 0,Y 122.108,Z 316.802,A -85,B 0,C 180,E1 -25633.276,E2 -25633.276} C_VEL
LIN {X 0,Y 120.897,Z 319.125,A -85,B 0,C 180,E1 -25636.555,E2 -25636.555} C_VEL
LIN {X 0,Y 119.987,Z 320.864,A -85,B 0,C 180,E1 -25639.88,E2 -25639.88} C_VEL
LIN {X 0,Y 119.441,Z 322.109,A -85,B 0,C 180,E1 -25643.242,E2 -25643.242} C_VEL
LIN {X 0,Y 119.225,Z 322.882,A -85,B 0,C 180,E1 -25646.621,E2 -25646.621} C_VEL
LIN {X 0,Y 119.278,Z 323.175,A -85,B 0,C 180,E1 -25650.001,E2 -25650.001} C_VEL
LIN {X 0,Y 119.226,Z 322.869,A -85,B 0,C 180,E1 -25653.38,E2 -25653.38} C_VEL
LIN {X 0,Y 119.439,Z 322.072,A -85,B 0,C 180,E1 -25656.759,E2 -25656.759} C_VEL
LIN {X 0,Y 119.974,Z 320.802,A -85,B 0,C 180,E1 -25660.122,E2 -25660.122} C_VEL
LIN {X 0,Y 121.397,Z 317.879,A -85,B 0,C 180,E1 -25665.102,E2 -25665.102} C_VEL
LIN {X 0,Y 122.842,Z 315.217,A -85,B 0,C 180,E1 -25668.341,E2 -25668.341} C_VEL
LIN {X 0,Y 125.639,Z 310.021,A -85,B 0,C 180,E1 -25673.053,E2 -25673.053} C_VEL
LIN {X 0,Y 129.324,Z 303.168,A -85,B 0,C 180,E1 -25677.512,E2 -25677.512} C_VEL
LIN {X 0,Y 132.943,Z 295.685,A -85,B 0,C 180,E1 -25681.027,E2 -25681.027} C_VEL
LIN {X 0,Y 136.191,Z 288.305,A -85,B 0,C 180,E1 -25683.694,E2 -25683.694} C_VEL
LIN {X 0,Y 139.235,Z 280.504,A -85,B 0,C 180,E1 -25685.892,E2 -25685.892} C_VEL
LIN {X 0,Y 142.212,Z 271.552,A -85,B 0,C 180,E1 -25687.848,E2 -25687.848} C_VEL
LIN {X 0,Y 145.184,Z 260.128,A -85,B 0,C 180,E1 -25689.68,E2 -25689.68} C_VEL
LIN {X 0,Y 147.279,Z 249.56,A -85,B 0,C 180,E1 -25690.785,E2 -25690.785} C_VEL
LIN {X 0,Y 148.446,Z 240.683,A -85,B 0,C 180,E1 -25691.426,E2 -25691.426} C_VEL
LIN {X 0,Y 149.529,Z 225.756,A -85,B 0,C 180,E1 -25692.117,E2 -25692.117} C_VEL
LIN {X 0,Y 149.199,Z 222.697,A -85,B 0,C 180,E1 -25692.426,E2 -25692.426} C_VEL
LIN {X 0,Y 147.524,Z 219.025,A -85,B 0,C 180,E1 -25693.259,E2 -25693.259} C_VEL
LIN {X 0,Y 141.812,Z 211.24,A -85,B 0,C 180,E1 -25696.011,E2 -25696.011} C_VEL
LIN {X 0,Y 141.07,Z 209.571,A -85,B 0,C 180,E1 -25696.443,E2 -25696.443} C_VEL
LIN {X 0,Y 136.991,Z 200.154,A -85,B 0,C 180,E1 -25698.988,E2 -25698.988} C_VEL
LIN {X 0,Y 132.166,Z 192.36,A -85,B 0,C 180,E1 -25702.11,E2 -25702.11} C_VEL
LIN {X 0,Y 129.097,Z 188.031,A -85,B 0,C 180,E1 -25704.287,E2 -25704.287} C_VEL
LIN {X 0,Y 126.364,Z 184.157,A -85,B 0,C 180,E1 -25706.425,E2 -25706.425} C_VEL
LIN {X 0,Y 123.945,Z 180.934,A -85,B 0,C 180,E1 -25708.485,E2 -25708.485} C_VEL
LIN {X 0,Y 123.117,Z 179.731,A -85,B 0,C 180,E1 -25709.249,E2 -25709.249} C_VEL
LIN {X 0,Y 120.638,Z 177.074,A -85,B 0,C 180,E1 -25711.6,E2 -25711.6} C_VEL
LIN {X 0,Y 119.331,Z 174.709,A -85,B 0,C 180,E1 -25713.08,E2 -25713.08} C_VEL
LIN {X 0,Y 116.597,Z 172.696,A -85,B 0,C 180,E1 -25716.137,E2 -25716.137} C_VEL
LIN {X 0,Y 115.086,Z 169.63,A -85,B 0,C 180,E1 -25718.741,E2 -25718.741} C_VEL
LIN {X 0,Y 114.993,Z 169.007,A -85,B 0,C 180,E1 -25720.358,E2 -25720.358} C_VEL
LIN {X 0,Y 115.254,Z 168.907,A -85,B 0,C 180,E1 -25727.333,E2 -25727.333} C_VEL
LIN {X 0,Y 115.37,Z 168.909,A -85,B 0,C 180,E1 -25733.002,E2 -25733.002} C_VEL
LIN {X 0,Y 115.995,Z 168.803,A -85,B 0,C 180,E1 -25740,E2 -25740} C_VEL
LIN {X 0,Y 115.385,Z 168.888,A -85,B 0,C 180,E1 -25746.997,E2 -25746.997} C_VEL
LIN {X 0,Y 115.307,Z 168.921,A -85,B 0,C 180,E1 -25752.783,E2 -25752.783} C_VEL
LIN {X 0,Y 115.032,Z 169.083,A -85,B 0,C 180,E1 -25760.567,E2 -25760.567} C_VEL
LIN {X 0,Y 115.222,Z 170.104,A -85,B 0,C 180,E1 -25762.066,E2 -25762.066} C_VEL
LIN {X 0,Y 116.757,Z 172.94,A -85,B 0,C 180,E1 -25764.374,E2 -25764.374} C_VEL
LIN {X 0,Y 119.636,Z 175.121,A -85,B 0,C 180,E1 -25767.557,E2 -25767.557} C_VEL
LIN {X 0,Y 121.363,Z 178.101,A -85,B 0,C 180,E1 -25769.445,E2 -25769.445} C_VEL
LIN {X 0,Y 123.649,Z 180.338,A -85,B 0,C 180,E1 -25771.526,E2 -25771.526} C_VEL
LIN {X 0,Y 125.997,Z 183.8,A -85,B 0,C 180,E1 -25773.588,E2 -25773.588} C_VEL
LIN {X 0,Y 127.279,Z 185.362,A -85,B 0,C 180,E1 -25774.605,E2 -25774.605} C_VEL
LIN {X 0,Y 131.204,Z 191.114,A -85,B 0,C 180,E1 -25777.54,E2 -25777.54} C_VEL
LIN {X 0,Y 135.344,Z 197.408,A -85,B 0,C 180,E1 -25780.287,E2 -25780.287} C_VEL
LIN {X 0,Y 140.789,Z 206.851,A -85,B 0,C 180,E1 -25783.539,E2 -25783.539} C_VEL
LIN {X 0,Y 144.597,Z 214.898,A -85,B 0,C 180,E1 -25785.664,E2 -25785.664} C_VEL
LIN {X 0,Y 144.977,Z 216.355,A -85,B 0,C 180,E1 -25785.91,E2 -25785.91} C_VEL
LIN {X 0,Y 143.358,Z 237.346,A -85,B 0,C 180,E1 -25786.853,E2 -25786.853} C_VEL
LIN {X 0,Y 141.84,Z 248.233,A -85,B 0,C 180,E1 -25787.714,E2 -25787.714} C_VEL
LIN {X 0,Y 139.533,Z 259.153,A -85,B 0,C 180,E1 -25789.096,E2 -25789.096} C_VEL
LIN {X 0,Y 136.813,Z 268.852,A -85,B 0,C 180,E1 -25790.817,E2 -25790.817} C_VEL
LIN {X 0,Y 134.241,Z 276.311,A -85,B 0,C 180,E1 -25792.51,E2 -25792.51} C_VEL
LIN {X 0,Y 131.063,Z 284.217,A -85,B 0,C 180,E1 -25794.798,E2 -25794.798} C_VEL
LIN {X 0,Y 127.68,Z 291.591,A -85,B 0,C 180,E1 -25797.542,E2 -25797.542} C_VEL
LIN {X 0,Y 123.835,Z 299.061,A -85,B 0,C 180,E1 -25801.157,E2 -25801.157} C_VEL
LIN {X 0,Y 119.936,Z 305.902,A -85,B 0,C 180,E1 -25805.783,E2 -25805.783} C_VEL
LIN {X 0,Y 116.82,Z 311.075,A -85,B 0,C 180,E1 -25810.677,E2 -25810.677} C_VEL
LIN {X 0,Y 115.175,Z 313.726,A -85,B 0,C 180,E1 -25814.062,E2 -25814.062} C_VEL
LIN {X 0,Y 113.451,Z 316.627,A -85,B 0,C 180,E1 -25819.289,E2 -25819.289} C_VEL
LIN {X 0,Y 112.748,Z 317.89,A -85,B 0,C 180,E1 -25822.838,E2 -25822.838} C_VEL
LIN {X 0,Y 112.288,Z 318.684,A -85,B 0,C 180,E1 -25826.411,E2 -25826.411} C_VEL
LIN {X 0,Y 112.208,Z 318.986,A -85,B 0,C 180,E1 -25829.999,E2 -25829.999} C_VEL
LIN {X 0,Y 112.287,Z 318.705,A -85,B 0,C 180,E1 -25833.588,E2 -25833.588} C_VEL
LIN {X 0,Y 112.717,Z 317.952,A -85,B 0,C 180,E1 -25837.163,E2 -25837.163} C_VEL
LIN {X 0,Y 113.382,Z 316.732,A -85,B 0,C 180,E1 -25840.716,E2 -25840.716} C_VEL
LIN {X 0,Y 115.164,Z 313.873,A -85,B 0,C 180,E1 -25845.938,E2 -25845.938} C_VEL
LIN {X 0,Y 116.765,Z 311.269,A -85,B 0,C 180,E1 -25849.331,E2 -25849.331} C_VEL
LIN {X 0,Y 119.89,Z 306.148,A -85,B 0,C 180,E1 -25854.225,E2 -25854.225} C_VEL
LIN {X 0,Y 123.07,Z 300.637,A -85,B 0,C 180,E1 -25858.106,E2 -25858.106} C_VEL
LIN {X 0,Y 126.781,Z 293.705,A -85,B 0,C 180,E1 -25861.777,E2 -25861.777} C_VEL
LIN {X 0,Y 130.552,Z 285.746,A -85,B 0,C 180,E1 -25864.887,E2 -25864.887} C_VEL
LIN {X 0,Y 133.781,Z 278.154,A -85,B 0,C 180,E1 -25867.166,E2 -25867.166} C_VEL
LIN {X 0,Y 136.699,Z 269.768,A -85,B 0,C 180,E1 -25869.17,E2 -25869.17} C_VEL
LIN {X 0,Y 139.213,Z 261.272,A -85,B 0,C 180,E1 -25870.715,E2 -25870.715} C_VEL
LIN {X 0,Y 141.322,Z 252.064,A -85,B 0,C 180,E1 -25871.997,E2 -25871.997} C_VEL
LIN {X 0,Y 143.251,Z 240.593,A -85,B 0,C 180,E1 -25873.101,E2 -25873.101} C_VEL
LIN {X 0,Y 144.541,Z 225.127,A -85,B 0,C 180,E1 -25873.905,E2 -25873.905} C_VEL
LIN {X 0,Y 145.049,Z 215.962,A -85,B 0,C 180,E1 -25874.331,E2 -25874.331} C_VEL
LIN {X 0,Y 142.608,Z 210.295,A -85,B 0,C 180,E1 -25875.7,E2 -25875.7} C_VEL
LIN {X 0,Y 138.128,Z 201.992,A -85,B 0,C 180,E1 -25878.278,E2 -25878.278} C_VEL
LIN {X 0,Y 133.945,Z 195.189,A -85,B 0,C 180,E1 -25880.899,E2 -25880.899} C_VEL
LIN {X 0,Y 129.568,Z 188.565,A -85,B 0,C 180,E1 -25883.963,E2 -25883.963} C_VEL
LIN {X 0,Y 126.478,Z 184.29,A -85,B 0,C 180,E1 -25886.37,E2 -25886.37} C_VEL
LIN {X 0,Y 123.905,Z 180.793,A -85,B 0,C 180,E1 -25888.591,E2 -25888.591} C_VEL
LIN {X 0,Y 123.177,Z 179.761,A -85,B 0,C 180,E1 -25889.268,E2 -25889.268} C_VEL
LIN {X 0,Y 120.708,Z 177.204,A -85,B 0,C 180,E1 -25891.622,E2 -25891.622} C_VEL
LIN {X 0,Y 119.426,Z 174.786,A -85,B 0,C 180,E1 -25893.102,E2 -25893.102} C_VEL
LIN {X 0,Y 116.536,Z 172.632,A -85,B 0,C 180,E1 -25896.394,E2 -25896.394} C_VEL
LIN {X 0,Y 115.099,Z 169.607,A -85,B 0,C 180,E1 -25898.977,E2 -25898.977} C_VEL
LIN {X 0,Y 114.998,Z 168.985,A -85,B 0,C 180,E1 -25901.285,E2 -25901.285} C_VEL
LIN {X 0,Y 115.304,Z 168.923,A -85,B 0,C 180,E1 -25907.217,E2 -25907.217} C_VEL
LIN {X 0,Y 115.382,Z 168.888,A -85,B 0,C 180,E1 -25913.002,E2 -25913.002} C_VEL
LIN {X 0,Y 115.995,Z 168.804,A -85,B 0,C 180,E1 -25920,E2 -25920} C_VEL
LIN {X 0,Y 115.389,Z 168.906,A -85,B 0,C 180,E1 -25926.996,E2 -25926.996} C_VEL
LIN {X 0,Y 115.283,Z 168.904,A -85,B 0,C 180,E1 -25932.738,E2 -25932.738} C_VEL
LIN {X 0,Y 115.045,Z 169.184,A -85,B 0,C 180,E1 -25940.098,E2 -25940.098} C_VEL
LIN {X 0,Y 115.27,Z 170.304,A -85,B 0,C 180,E1 -25941.458,E2 -25941.458} C_VEL
LIN {X 0,Y 117.037,Z 173.201,A -85,B 0,C 180,E1 -25944.039,E2 -25944.039} C_VEL
LIN {X 0,Y 119.578,Z 175.005,A -85,B 0,C 180,E1 -25946.86,E2 -25946.86} C_VEL
LIN {X 0,Y 121.608,Z 178.358,A -85,B 0,C 180,E1 -25949.084,E2 -25949.084} C_VEL
LIN {X 0,Y 123.696,Z 180.346,A -85,B 0,C 180,E1 -25950.991,E2 -25950.991} C_VEL
LIN {X 0,Y 126.13,Z 183.931,A -85,B 0,C 180,E1 -25953.144,E2 -25953.144} C_VEL
LIN {X 0,Y 127.465,Z 185.666,A -85,B 0,C 180,E1 -25954.219,E2 -25954.219} C_VEL
LIN {X 0,Y 130.896,Z 190.523,A -85,B 0,C 180,E1 -25956.798,E2 -25956.798} C_VEL
LIN {X 0,Y 136.032,Z 198.438,A -85,B 0,C 180,E1 -25960.226,E2 -25960.226} C_VEL
LIN {X 0,Y 138.779,Z 203.842,A -85,B 0,C 180,E1 -25961.954,E2 -25961.954} C_VEL
LIN {X 0,Y 143.146,Z 214.85,A -85,B 0,C 180,E1 -25964.631,E2 -25964.631} C_VEL
LIN {X 0,Y 144.675,Z 219.144,A -85,B 0,C 180,E1 -25965.531,E2 -25965.531} C_VEL
LIN {X 0,Y 144.682,Z 223.227,A -85,B 0,C 180,E1 -25965.811,E2 -25965.811} C_VEL
LIN {X 0,Y 143.198,Z 242.204,A -85,B 0,C 180,E1 -25966.698,E2 -25966.698} C_VEL
LIN {X 0,Y 141.434,Z 253.518,A -85,B 0,C 180,E1 -25967.627,E2 -25967.627} C_VEL
LIN {X 0,Y 139.05,Z 263.72,A -85,B 0,C 180,E1 -25968.925,E2 -25968.925} C_VEL
LIN {X 0,Y 136.492,Z 272.38,A -85,B 0,C 180,E1 -25970.42,E2 -25970.42} C_VEL
LIN {X 0,Y 133.79,Z 280.166,A -85,B 0,C 180,E1 -25972.177,E2 -25972.177} C_VEL
LIN {X 0,Y 130.83,Z 287.466,A -85,B 0,C 180,E1 -25974.255,E2 -25974.255} C_VEL
LIN {X 0,Y 127.706,Z 294.111,A -85,B 0,C 180,E1 -25976.612,E2 -25976.612} C_VEL
LIN {X 0,Y 124.563,Z 300.425,A -85,B 0,C 180,E1 -25979.484,E2 -25979.484} C_VEL
LIN {X 0,Y 121.667,Z 305.669,A -85,B 0,C 180,E1 -25982.477,E2 -25982.477} C_VEL
LIN {X 0,Y 119.138,Z 310.042,A -85,B 0,C 180,E1 -25985.612,E2 -25985.612} C_VEL
LIN {X 0,Y 116.132,Z 315.206,A -85,B 0,C 180,E1 -25990.559,E2 -25990.559} C_VEL
LIN {X 0,Y 113.989,Z 318.998,A -85,B 0,C 180,E1 -25995.723,E2 -25995.723} C_VEL
LIN {X 0,Y 112.988,Z 320.736,A -85,B 0,C 180,E1 -25999.246,E2 -25999.246} C_VEL
LIN {X 0,Y 112.377,Z 321.981,A -85,B 0,C 180,E1 -26002.816,E2 -26002.816} C_VEL
LIN {X 0,Y 112.136,Z 322.753,A -85,B 0,C 180,E1 -26006.408,E2 -26006.408} C_VEL
LIN {X 0,Y 112.197,Z 323.046,A -85,B 0,C 180,E1 -26010.001,E2 -26010.001} C_VEL
LIN {X 0,Y 112.136,Z 322.741,A -85,B 0,C 180,E1 -26013.594,E2 -26013.594} C_VEL
LIN {X 0,Y 112.375,Z 321.943,A -85,B 0,C 180,E1 -26017.186,E2 -26017.186} C_VEL
LIN {X 0,Y 112.973,Z 320.672,A -85,B 0,C 180,E1 -26020.757,E2 -26020.757} C_VEL
LIN {X 0,Y 114.542,Z 317.75,A -85,B 0,C 180,E1 -26026.029,E2 -26026.029} C_VEL
LIN {X 0,Y 116.115,Z 315.088,A -85,B 0,C 180,E1 -26029.445,E2 -26029.445} C_VEL
LIN {X 0,Y 119.125,Z 309.89,A -85,B 0,C 180,E1 -26034.393,E2 -26034.393} C_VEL
LIN {X 0,Y 123.067,Z 303.037,A -85,B 0,C 180,E1 -26039.04,E2 -26039.04} C_VEL
LIN {X 0,Y 126.892,Z 295.554,A -85,B 0,C 180,E1 -26042.685,E2 -26042.685} C_VEL
LIN {X 0,Y 130.353,Z 288.174,A -85,B 0,C 180,E1 -26045.422,E2 -26045.422} C_VEL
LIN {X 0,Y 133.182,Z 281.336,A -85,B 0,C 180,E1 -26047.426,E2 -26047.426} C_VEL
LIN {X 0,Y 135.906,Z 273.708,A -85,B 0,C 180,E1 -26049.211,E2 -26049.211} C_VEL
LIN {X 0,Y 138.479,Z 265.007,A -85,B 0,C 180,E1 -26050.801,E2 -26050.801} C_VEL
LIN {X 0,Y 140.921,Z 255.011,A -85,B 0,C 180,E1 -26052.117,E2 -26052.117} C_VEL
LIN {X 0,Y 143.043,Z 242.349,A -85,B 0,C 180,E1 -26053.197,E2 -26053.197} C_VEL
LIN {X 0,Y 144.541,Z 222.622,A -85,B 0,C 180,E1 -26054.132,E2 -26054.132} C_VEL
LIN {X 0,Y 144.42,Z 218.6,A -85,B 0,C 180,E1 -26054.452,E2 -26054.452} C_VEL
LIN {X 0,Y 141.07,Z 209.571,A -85,B 0,C 180,E1 -26056.443,E2 -26056.443} C_VEL
LIN {X 0,Y 139.616,Z 206.595,A -85,B 0,C 180,E1 -26057.291,E2 -26057.291} C_VEL
LIN {X 0,Y 136.768,Z 203.078,A -85,B 0,C 180,E1 -26058.866,E2 -26058.866} C_VEL
LIN {X 0,Y 131.375,Z 198.74,A -85,B 0,C 180,E1 -26061.996,E2 -26061.996} C_VEL
LIN {X 0,Y 126.402,Z 194.183,A -85,B 0,C 180,E1 -26065.407,E2 -26065.407} C_VEL
LIN {X 0,Y 125.575,Z 193.023,A -85,B 0,C 180,E1 -26066.071,E2 -26066.071} C_VEL
LIN {X 0,Y 123.469,Z 189.953,A -85,B 0,C 180,E1 -26067.869,E2 -26067.869} C_VEL
LIN {X 0,Y 120.673,Z 185.902,A -85,B 0,C 180,E1 -26070.511,E2 -26070.511} C_VEL
LIN {X 0,Y 118.187,Z 182.976,A -85,B 0,C 180,E1 -26073.084,E2 -26073.084} C_VEL
LIN {X 0,Y 117.116,Z 181.166,A -85,B 0,C 180,E1 -26074.377,E2 -26074.377} C_VEL
LIN {X 0,Y 114.523,Z 178.874,A -85,B 0,C 180,E1 -26077.573,E2 -26077.573} C_VEL
LIN {X 0,Y 113.025,Z 175.926,A -85,B 0,C 180,E1 -26080.002,E2 -26080.002} C_VEL
LIN {X 0,Y 109.916,Z 173.771,A -85,B 0,C 180,E1 -26085.564,E2 -26085.564} C_VEL
LIN {X 0,Y 108.414,Z 170.603,A -85,B 0,C 180,E1 -26090.674,E2 -26090.674} C_VEL
LIN {X 0,Y 108.371,Z 169.821,A -85,B 0,C 180,E1 -26095.118,E2 -26095.118} C_VEL
LIN {X 0,Y 108.945,Z 169.698,A -85,B 0,C 180,E1 -26100,E2 -26100} C_VEL
LIN {X 0,Y 108.361,Z 170.251,A -85,B 0,C 180,E1 -26108.391,E2 -26108.391} C_VEL
LIN {X 0,Y 108.648,Z 171.261,A -85,B 0,C 180,E1 -26110.954,E2 -26110.954} C_VEL
LIN {X 0,Y 110.354,Z 174.271,A -85,B 0,C 180,E1 -26115.704,E2 -26115.704} C_VEL
LIN {X 0,Y 113.06,Z 175.941,A -85,B 0,C 180,E1 -26120.348,E2 -26120.348} C_VEL
LIN {X 0,Y 114.699,Z 179.136,A -85,B 0,C 180,E1 -26122.978,E2 -26122.978} C_VEL
LIN {X 0,Y 117.186,Z 181.294,A -85,B 0,C 180,E1 -26126.012,E2 -26126.012} C_VEL
LIN {X 0,Y 119.904,Z 185.224,A -85,B 0,C 180,E1 -26129.054,E2 -26129.054} C_VEL
LIN {X 0,Y 121.286,Z 186.777,A -85,B 0,C 180,E1 -26130.395,E2 -26130.395} C_VEL
LIN {X 0,Y 123.844,Z 190.338,A -85,B 0,C 180,E1 -26132.744,E2 -26132.744} C_VEL
LIN {X 0,Y 128.06,Z 196.656,A -85,B 0,C 180,E1 -26136.18,E2 -26136.18} C_VEL
LIN {X 0,Y 133.059,Z 204.71,A -85,B 0,C 180,E1 -26139.716,E2 -26139.716} C_VEL
LIN {X 0,Y 137.686,Z 213.456,A -85,B 0,C 180,E1 -26142.657,E2 -26142.657} C_VEL
LIN {X 0,Y 139.796,Z 218.026,A -85,B 0,C 180,E1 -26143.926,E2 -26143.926} C_VEL
LIN {X 0,Y 138.189,Z 238.534,A -85,B 0,C 180,E1 -26144.913,E2 -26144.913} C_VEL
LIN {X 0,Y 136.217,Z 250.726,A -85,B 0,C 180,E1 -26145.982,E2 -26145.982} C_VEL
LIN {X 0,Y 133.867,Z 260.655,A -85,B 0,C 180,E1 -26147.335,E2 -26147.335} C_VEL
LIN {X 0,Y 131.268,Z 269.359,A -85,B 0,C 180,E1 -26148.942,E2 -26148.942} C_VEL
LIN {X 0,Y 128.684,Z 276.443,A -85,B 0,C 180,E1 -26150.587,E2 -26150.587} C_VEL
LIN {X 0,Y 125.335,Z 284.349,A -85,B 0,C 180,E1 -26152.929,E2 -26152.929} C_VEL
LIN {X 0,Y 121.764,Z 291.722,A -85,B 0,C 180,E1 -26155.753,E2 -26155.753} C_VEL
LIN {X 0,Y 117.671,Z 299.192,A -85,B 0,C 180,E1 -26159.491,E2 -26159.491} C_VEL
LIN {X 0,Y 113.507,Z 306.032,A -85,B 0,C 180,E1 -26164.314,E2 -26164.314} C_VEL
LIN {X 0,Y 110.133,Z 311.205,A -85,B 0,C 180,E1 -26169.452,E2 -26169.452} C_VEL
LIN {X 0,Y 108.373,Z 313.855,A -85,B 0,C 180,E1 -26173.032,E2 -26173.032} C_VEL
LIN {X 0,Y 106.475,Z 316.757,A -85,B 0,C 180,E1 -26178.578,E2 -26178.578} C_VEL
LIN {X 0,Y 105.718,Z 318.018,A -85,B 0,C 180,E1 -26182.359,E2 -26182.359} C_VEL
LIN {X 0,Y 105.23,Z 318.813,A -85,B 0,C 180,E1 -26186.17,E2 -26186.17} C_VEL
LIN {X 0,Y 105.114,Z 319.114,A -85,B 0,C 180,E1 -26189.999,E2 -26189.999} C_VEL
LIN {X 0,Y 105.229,Z 318.833,A -85,B 0,C 180,E1 -26193.829,E2 -26193.829} C_VEL
LIN {X 0,Y 105.667,Z 318.08,A -85,B 0,C 180,E1 -26197.643,E2 -26197.643} C_VEL
LIN {X 0,Y 106.422,Z 316.86,A -85,B 0,C 180,E1 -26201.426,E2 -26201.426} C_VEL
LIN {X 0,Y 108.361,Z 314,A -85,B 0,C 180,E1 -26206.968,E2 -26206.968} C_VEL
LIN {X 0,Y 110.079,Z 311.396,A -85,B 0,C 180,E1 -26210.557,E2 -26210.557} C_VEL
LIN {X 0,Y 113.461,Z 306.275,A -85,B 0,C 180,E1 -26215.695,E2 -26215.695} C_VEL
LIN {X 0,Y 116.861,Z 300.764,A -85,B 0,C 180,E1 -26219.745,E2 -26219.745} C_VEL
LIN {X 0,Y 120.818,Z 293.831,A -85,B 0,C 180,E1 -26223.546,E2 -26223.546} C_VEL
LIN {X 0,Y 124.804,Z 285.871,A -85,B 0,C 180,E1 -26226.748,E2 -26226.748} C_VEL
LIN {X 0,Y 128.2,Z 278.279,A -85,B 0,C 180,E1 -26229.081,E2 -26229.081} C_VEL
LIN {X 0,Y 131.169,Z 270.237,A -85,B 0,C 180,E1 -26231.049,E2 -26231.049} C_VEL
LIN {X 0,Y 133.873,Z 261.558,A -85,B 0,C 180,E1 -26232.667,E2 -26232.667} C_VEL
LIN {X 0,Y 136.016,Z 252.771,A -85,B 0,C 180,E1 -26233.918,E2 -26233.918} C_VEL
LIN {X 0,Y 137.773,Z 243.056,A -85,B 0,C 180,E1 -26234.914,E2 -26234.914} C_VEL
LIN {X 0,Y 139.094,Z 231.301,A -85,B 0,C 180,E1 -26235.664,E2 -26235.664} C_VEL
LIN {X 0,Y 139.928,Z 218.07,A -85,B 0,C 180,E1 -26236.27,E2 -26236.27} C_VEL
LIN {X 0,Y 135.909,Z 209.793,A -85,B 0,C 180,E1 -26238.725,E2 -26238.725} C_VEL
LIN {X 0,Y 131.379,Z 201.743,A -85,B 0,C 180,E1 -26241.73,E2 -26241.73} C_VEL
LIN {X 0,Y 126.232,Z 193.834,A -85,B 0,C 180,E1 -26245.584,E2 -26245.584} C_VEL
LIN {X 0,Y 123.422,Z 189.831,A -85,B 0,C 180,E1 -26247.974,E2 -26247.974} C_VEL
LIN {X 0,Y 120.734,Z 185.951,A -85,B 0,C 180,E1 -26250.542,E2 -26250.542} C_VEL
LIN {X 0,Y 118.193,Z 182.969,A -85,B 0,C 180,E1 -26253.206,E2 -26253.206} C_VEL
LIN {X 0,Y 117.207,Z 181.23,A -85,B 0,C 180,E1 -26254.422,E2 -26254.422} C_VEL
LIN {X 0,Y 114.584,Z 178.935,A -85,B 0,C 180,E1 -26257.702,E2 -26257.702} C_VEL
LIN {X 0,Y 112.911,Z 175.857,A -85,B 0,C 180,E1 -26260.454,E2 -26260.454} C_VEL
LIN {X 0,Y 109.992,Z 173.821,A -85,B 0,C 180,E1 -26265.891,E2 -26265.891} C_VEL
LIN {X 0,Y 108.445,Z 170.565,A -85,B 0,C 180,E1 -26271.615,E2 -26271.615} C_VEL
LIN {X 0,Y 108.472,Z 169.874,A -85,B 0,C 180,E1 -26276.285,E2 -26276.285} C_VEL
LIN {X 0,Y 108.945,Z 169.724,A -85,B 0,C 180,E1 -26280,E2 -26280} C_VEL
LIN {X 0,Y 108.428,Z 170.337,A -85,B 0,C 180,E1 -26287.448,E2 -26287.448} C_VEL
LIN {X 0,Y 108.961,Z 171.971,A -85,B 0,C 180,E1 -26290.921,E2 -26290.921} C_VEL
LIN {X 0,Y 110.781,Z 174.625,A -85,B 0,C 180,E1 -26295.641,E2 -26295.641} C_VEL
LIN {X 0,Y 113.155,Z 176.15,A -85,B 0,C 180,E1 -26299.738,E2 -26299.738} C_VEL
LIN {X 0,Y 115.066,Z 179.545,A -85,B 0,C 180,E1 -26302.766,E2 -26302.766} C_VEL
LIN {X 0,Y 117.508,Z 181.606,A -85,B 0,C 180,E1 -26305.726,E2 -26305.726} C_VEL
LIN {X 0,Y 119.862,Z 185.166,A -85,B 0,C 180,E1 -26308.402,E2 -26308.402} C_VEL
LIN {X 0,Y 121.34,Z 186.773,A -85,B 0,C 180,E1 -26309.849,E2 -26309.849} C_VEL
LIN {X 0,Y 123.862,Z 190.34,A -85,B 0,C 180,E1 -26312.196,E2 -26312.196} C_VEL
LIN {X 0,Y 127.749,Z 196.088,A -85,B 0,C 180,E1 -26315.406,E2 -26315.406} C_VEL
LIN {X 0,Y 131.895,Z 202.631,A -85,B 0,C 180,E1 -26318.42,E2 -26318.42} C_VEL
LIN {X 0,Y 133.957,Z 206.579,A -85,B 0,C 180,E1 -26319.839,E2 -26319.839} C_VEL
LIN {X 0,Y 138.096,Z 216.992,A -85,B 0,C 180,E1 -26322.636,E2 -26322.636} C_VEL
LIN {X 0,Y 139.717,Z 221.621,A -85,B 0,C 180,E1 -26323.688,E2 -26323.688} C_VEL
LIN {X 0,Y 138.251,Z 241.043,A -85,B 0,C 180,E1 -26324.629,E2 -26324.629} C_VEL
LIN {X 0,Y 136.429,Z 252.712,A -85,B 0,C 180,E1 -26325.545,E2 -26325.545} C_VEL
LIN {X 0,Y 133.79,Z 263.598,A -85,B 0,C 180,E1 -26326.931,E2 -26326.931} C_VEL
LIN {X 0,Y 131.105,Z 272.251,A -85,B 0,C 180,E1 -26328.443,E2 -26328.443} C_VEL
LIN {X 0,Y 128.261,Z 280.042,A -85,B 0,C 180,E1 -26330.233,E2 -26330.233} C_VEL
LIN {X 0,Y 125.139,Z 287.341,A -85,B 0,C 180,E1 -26332.357,E2 -26332.357} C_VEL
LIN {X 0,Y 121.844,Z 293.986,A -85,B 0,C 180,E1 -26334.775,E2 -26334.775} C_VEL
LIN {X 0,Y 118.489,Z 300.298,A -85,B 0,C 180,E1 -26337.737,E2 -26337.737} C_VEL
LIN {X 0,Y 115.409,Z 305.542,A -85,B 0,C 180,E1 -26340.846,E2 -26340.846} C_VEL
LIN {X 0,Y 112.699,Z 309.915,A -85,B 0,C 180,E1 -26344.119,E2 -26344.119} C_VEL
LIN {X 0,Y 109.454,Z 315.079,A -85,B 0,C 180,E1 -26349.321,E2 -26349.321} C_VEL
LIN {X 0,Y 107.116,Z 318.87,A -85,B 0,C 180,E1 -26354.786,E2 -26354.786} C_VEL
LIN {X 0,Y 106.017,Z 320.608,A -85,B 0,C 180,E1 -26358.53,E2 -26358.53} C_VEL
LIN {X 0,Y 105.323,Z 321.852,A -85,B 0,C 180,E1 -26362.332,E2 -26362.332} C_VEL
LIN {X 0,Y 105.047,Z 322.625,A -85,B 0,C 180,E1 -26366.165,E2 -26366.165} C_VEL
LIN {X 0,Y 105.104,Z 322.918,A -85,B 0,C 180,E1 -26370.001,E2 -26370.001} C_VEL
LIN {X 0,Y 105.047,Z 322.612,A -85,B 0,C 180,E1 -26373.837,E2 -26373.837} C_VEL
LIN {X 0,Y 105.32,Z 321.814,A -85,B 0,C 180,E1 -26377.67,E2 -26377.67} C_VEL
LIN {X 0,Y 106.002,Z 320.543,A -85,B 0,C 180,E1 -26381.474,E2 -26381.474} C_VEL
LIN {X 0,Y 107.727,Z 317.62,A -85,B 0,C 180,E1 -26387.073,E2 -26387.073} C_VEL
LIN {X 0,Y 109.44,Z 314.958,A -85,B 0,C 180,E1 -26390.684,E2 -26390.684} C_VEL
LIN {X 0,Y 112.685,Z 309.76,A -85,B 0,C 180,E1 -26395.887,E2 -26395.887} C_VEL
LIN {X 0,Y 116.911,Z 302.907,A -85,B 0,C 180,E1 -26400.729,E2 -26400.729} C_VEL
LIN {X 0,Y 120.966,Z 295.422,A -85,B 0,C 180,E1 -26404.505,E2 -26404.505} C_VEL
LIN {X 0,Y 124.636,Z 288.042,A -85,B 0,C 180,E1 -26407.314,E2 -26407.314} C_VEL
LIN {X 0,Y 127.714,Z 280.97,A -85,B 0,C 180,E1 -26409.425,E2 -26409.425} C_VEL
LIN {X 0,Y 130.592,Z 273.272,A -85,B 0,C 180,E1 -26411.244,E2 -26411.244} C_VEL
LIN {X 0,Y 133.188,Z 264.871,A -85,B 0,C 180,E1 -26412.796,E2 -26412.796} C_VEL
LIN {X 0,Y 135.623,Z 255.423,A -85,B 0,C 180,E1 -26414.058,E2 -26414.058} C_VEL
LIN {X 0,Y 137.778,Z 243.922,A -85,B 0,C 180,E1 -26415.102,E2 -26415.102} C_VEL
LIN {X 0,Y 139.127,Z 228.643,A -85,B 0,C 180,E1 -26415.888,E2 -26415.888} C_VEL
LIN {X 0,Y 139.471,Z 221.216,A -85,B 0,C 180,E1 -26416.28,E2 -26416.28} C_VEL
LIN {X 0,Y 135.024,Z 209.255,A -85,B 0,C 180,E1 -26419.223,E2 -26419.223} C_VEL
LIN {X 0,Y 132.612,Z 204.005,A -85,B 0,C 180,E1 -26420.877,E2 -26420.877} C_VEL
LIN {X 0,Y 128.145,Z 196.785,A -85,B 0,C 180,E1 -26424.056,E2 -26424.056} C_VEL
LIN {X 0,Y 125.974,Z 193.577,A -85,B 0,C 180,E1 -26425.749,E2 -26425.749} C_VEL
LIN {X 0,Y 125.575,Z 193.023,A -85,B 0,C 180,E1 -26426.071,E2 -26426.071} C_VEL
LIN {X 0,Y 123.766,Z 191.377,A -85,B 0,C 180,E1 -26427.503,E2 -26427.503} C_VEL
LIN {X 0,Y 120.334,Z 190.71,A -85,B 0,C 180,E1 -26430.227,E2 -26430.227} C_VEL
LIN {X 0,Y 117.153,Z 190.135,A -85,B 0,C 180,E1 -26433.128,E2 -26433.128} C_VEL
LIN {X 0,Y 115.692,Z 188.612,A -85,B 0,C 180,E1 -26434.8,E2 -26434.8} C_VEL
LIN {X 0,Y 114.929,Z 187.567,A -85,B 0,C 180,E1 -26435.768,E2 -26435.768} C_VEL
LIN {X 0,Y 112.452,Z 184.93,A -85,B 0,C 180,E1 -26439.179,E2 -26439.179} C_VEL
LIN {X 0,Y 111.302,Z 182.562,A -85,B 0,C 180,E1 -26441.238,E2 -26441.238} C_VEL
LIN {X 0,Y 108.596,Z 180.497,A -85,B 0,C 180,E1 -26446.543,E2 -26446.543} C_VEL
LIN {X 0,Y 107.141,Z 177.412,A -85,B 0,C 180,E1 -26451.513,E2 -26451.513} C_VEL
LIN {X 0,Y 106.282,Z 176.565,A -85,B 0,C 180,E1 -26456.209,E2 -26456.209} C_VEL
LIN {X 0,Y 106.073,Z 176.304,A -85,B 0,C 180,E1 -26460.95,E2 -26460.95} C_VEL
LIN {X 0,Y 107.073,Z 177.308,A -85,B 0,C 180,E1 -26468.493,E2 -26468.493} C_VEL
LIN {X 0,Y 107.86,Z 179.093,A -85,B 0,C 180,E1 -26471.581,E2 -26471.581} C_VEL
LIN {X 0,Y 109.291,Z 181.284,A -85,B 0,C 180,E1 -26475.383,E2 -26475.383} C_VEL
LIN {X 0,Y 111.448,Z 182.853,A -85,B 0,C 180,E1 -26479.334,E2 -26479.334} C_VEL
LIN {X 0,Y 113.392,Z 186.251,A -85,B 0,C 180,E1 -26482.543,E2 -26482.543} C_VEL
LIN {X 0,Y 115.549,Z 188.396,A -85,B 0,C 180,E1 -26485.32,E2 -26485.32} C_VEL
LIN {X 0,Y 118.023,Z 191.86,A -85,B 0,C 180,E1 -26488.207,E2 -26488.207} C_VEL
LIN {X 0,Y 119.276,Z 193.667,A -85,B 0,C 180,E1 -26489.534,E2 -26489.534} C_VEL
LIN {X 0,Y 122.177,Z 197.902,A -85,B 0,C 180,E1 -26492.328,E2 -26492.328} C_VEL
LIN {X 0,Y 126.176,Z 204.104,A -85,B 0,C 180,E1 -26495.707,E2 -26495.707} C_VEL
LIN {X 0,Y 130.948,Z 212.493,A -85,B 0,C 180,E1 -26499.252,E2 -26499.252} C_VEL
LIN {X 0,Y 134.799,Z 220.405,A -85,B 0,C 180,E1 -26501.849,E2 -26501.849} C_VEL
LIN {X 0,Y 133.195,Z 239.323,A -85,B 0,C 180,E1 -26502.785,E2 -26502.785} C_VEL
LIN {X 0,Y 131.052,Z 251.569,A -85,B 0,C 180,E1 -26503.92,E2 -26503.92} C_VEL
LIN {X 0,Y 128.654,Z 261.098,A -85,B 0,C 180,E1 -26505.248,E2 -26505.248} C_VEL
LIN {X 0,Y 126.211,Z 268.905,A -85,B 0,C 180,E1 -26506.696,E2 -26506.696} C_VEL
LIN {X 0,Y 123.279,Z 276.576,A -85,B 0,C 180,E1 -26508.491,E2 -26508.491} C_VEL
LIN {X 0,Y 119.752,Z 284.48,A -85,B 0,C 180,E1 -26510.883,E2 -26510.883} C_VEL
LIN {X 0,Y 115.967,Z 291.853,A -85,B 0,C 180,E1 -26513.779,E2 -26513.779} C_VEL
LIN {X 0,Y 111.619,Z 299.322,A -85,B 0,C 180,E1 -26517.642,E2 -26517.642} C_VEL
LIN {X 0,Y 107.142,Z 306.162,A -85,B 0,C 180,E1 -26522.666,E2 -26522.666} C_VEL
LIN {X 0,Y 103.507,Z 311.335,A -85,B 0,C 180,E1 -26528.071,E2 -26528.071} C_VEL
LIN {X 0,Y 101.617,Z 313.984,A -85,B 0,C 180,E1 -26531.866,E2 -26531.866} C_VEL
LIN {X 0,Y 99.533,Z 316.886,A -85,B 0,C 180,E1 -26537.769,E2 -26537.769} C_VEL
LIN {X 0,Y 98.685,Z 318.147,A -85,B 0,C 180,E1 -26541.81,E2 -26541.81} C_VEL
LIN {X 0,Y 98.146,Z 318.941,A -85,B 0,C 180,E1 -26545.893,E2 -26545.893} C_VEL
LIN {X 0,Y 98.015,Z 319.243,A -85,B 0,C 180,E1 -26549.999,E2 -26549.999} C_VEL
LIN {X 0,Y 98.143,Z 318.961,A -85,B 0,C 180,E1 -26554.105,E2 -26554.105} C_VEL
LIN {X 0,Y 98.647,Z 318.208,A -85,B 0,C 180,E1 -26558.191,E2 -26558.191} C_VEL
LIN {X 0,Y 99.491,Z 316.988,A -85,B 0,C 180,E1 -26562.234,E2 -26562.234} C_VEL
LIN {X 0,Y 101.577,Z 314.128,A -85,B 0,C 180,E1 -26568.14,E2 -26568.14} C_VEL
LIN {X 0,Y 103.455,Z 311.523,A -85,B 0,C 180,E1 -26571.939,E2 -26571.939} C_VEL
LIN {X 0,Y 107.095,Z 306.402,A -85,B 0,C 180,E1 -26577.345,E2 -26577.345} C_VEL
LIN {X 0,Y 110.761,Z 300.89,A -85,B 0,C 180,E1 -26581.565,E2 -26581.565} C_VEL
LIN {X 0,Y 114.978,Z 293.957,A -85,B 0,C 180,E1 -26585.498,E2 -26585.498} C_VEL
LIN {X 0,Y 119.201,Z 285.996,A -85,B 0,C 180,E1 -26588.787,E2 -26588.787} C_VEL
LIN {X 0,Y 122.778,Z 278.403,A -85,B 0,C 180,E1 -26591.167,E2 -26591.167} C_VEL
LIN {X 0,Y 125.452,Z 271.639,A -85,B 0,C 180,E1 -26592.895,E2 -26592.895} C_VEL
LIN {X 0,Y 128.193,Z 263.57,A -85,B 0,C 180,E1 -26594.495,E2 -26594.495} C_VEL
LIN {X 0,Y 130.526,Z 255.007,A -85,B 0,C 180,E1 -26595.8,E2 -26595.8} C_VEL
LIN {X 0,Y 132.431,Z 245.717,A -85,B 0,C 180,E1 -26596.84,E2 -26596.84} C_VEL
LIN {X 0,Y 133.665,Z 236.839,A -85,B 0,C 180,E1 -26597.534,E2 -26597.534} C_VEL
LIN {X 0,Y 134.936,Z 220.521,A -85,B 0,C 180,E1 -26598.349,E2 -26598.349} C_VEL
LIN {X 0,Y 130.972,Z 212.406,A -85,B 0,C 180,E1 -26601.035,E2 -26601.035} C_VEL
LIN {X 0,Y 127.103,Z 205.6,A -85,B 0,C 180,E1 -26603.89,E2 -26603.89} C_VEL
LIN {X 0,Y 123.288,Z 199.498,A -85,B 0,C 180,E1 -26607.043,E2 -26607.043} C_VEL
LIN {X 0,Y 120.656,Z 195.591,A -85,B 0,C 180,E1 -26609.479,E2 -26609.479} C_VEL
LIN {X 0,Y 118.341,Z 192.152,A -85,B 0,C 180,E1 -26611.878,E2 -26611.878} C_VEL
LIN {X 0,Y 115.697,Z 188.593,A -85,B 0,C 180,E1 -26614.956,E2 -26614.956} C_VEL
LIN {X 0,Y 115.153,Z 187.691,A -85,B 0,C 180,E1 -26615.679,E2 -26615.679} C_VEL
LIN {X 0,Y 112.626,Z 185.121,A -85,B 0,C 180,E1 -26619.167,E2 -26619.167} C_VEL
LIN {X 0,Y 111.279,Z 182.566,A -85,B 0,C 180,E1 -26621.592,E2 -26621.592} C_VEL
LIN {X 0,Y 108.646,Z 180.47,A -85,B 0,C 180,E1 -26627.002,E2 -26627.002} C_VEL
LIN {X 0,Y 107.184,Z 177.395,A -85,B 0,C 180,E1 -26632.464,E2 -26632.464} C_VEL
LIN {X 0,Y 106.411,Z 176.366,A -85,B 0,C 180,E1 -26640,E2 -26640} C_VEL
LIN {X 0,Y 107.227,Z 177.46,A -85,B 0,C 180,E1 -26647.532,E2 -26647.532} C_VEL
LIN {X 0,Y 109.664,Z 181.582,A -85,B 0,C 180,E1 -26655.209,E2 -26655.209} C_VEL
LIN {X 0,Y 111.491,Z 182.842,A -85,B 0,C 180,E1 -26658.58,E2 -26658.58} C_VEL
LIN {X 0,Y 113.411,Z 186.198,A -85,B 0,C 180,E1 -26661.827,E2 -26661.827} C_VEL
LIN {X 0,Y 115.562,Z 188.259,A -85,B 0,C 180,E1 -26664.642,E2 -26664.642} C_VEL
LIN {X 0,Y 117.951,Z 191.742,A -85,B 0,C 180,E1 -26667.501,E2 -26667.501} C_VEL
LIN {X 0,Y 119.152,Z 193.335,A -85,B 0,C 180,E1 -26668.782,E2 -26668.782} C_VEL
LIN {X 0,Y 122.492,Z 198.311,A -85,B 0,C 180,E1 -26672.039,E2 -26672.039} C_VEL
LIN {X 0,Y 125.488,Z 202.87,A -85,B 0,C 180,E1 -26674.606,E2 -26674.606} C_VEL
LIN {X 0,Y 129.816,Z 210.372,A -85,B 0,C 180,E1 -26677.939,E2 -26677.939} C_VEL
LIN {X 0,Y 133.795,Z 220.914,A -85,B 0,C 180,E1 -26680.918,E2 -26680.918} C_VEL
LIN {X 0,Y 134.701,Z 223.685,A -85,B 0,C 180,E1 -26681.578,E2 -26681.578} C_VEL
LIN {X 0,Y 133.372,Z 240.931,A -85,B 0,C 180,E1 -26682.463,E2 -26682.463} C_VEL
LIN {X 0,Y 131.542,Z 252.185,A -85,B 0,C 180,E1 -26683.337,E2 -26683.337} C_VEL
LIN {X 0,Y 128.696,Z 263.475,A -85,B 0,C 180,E1 -26684.773,E2 -26684.773} C_VEL
LIN {X 0,Y 125.874,Z 272.127,A -85,B 0,C 180,E1 -26686.297,E2 -26686.297} C_VEL
LIN {X 0,Y 122.978,Z 279.685,A -85,B 0,C 180,E1 -26688.049,E2 -26688.049} C_VEL
LIN {X 0,Y 119.6,Z 287.216,A -85,B 0,C 180,E1 -26690.281,E2 -26690.281} C_VEL
LIN {X 0,Y 116.124,Z 293.86,A -85,B 0,C 180,E1 -26692.757,E2 -26692.757} C_VEL
LIN {X 0,Y 112.535,Z 300.172,A -85,B 0,C 180,E1 -26695.803,E2 -26695.803} C_VEL
LIN {X 0,Y 109.259,Z 305.415,A -85,B 0,C 180,E1 -26699.031,E2 -26699.031} C_VEL
LIN {X 0,Y 106.35,Z 309.788,A -85,B 0,C 180,E1 -26702.447,E2 -26702.447} C_VEL
LIN {X 0,Y 102.836,Z 314.951,A -85,B 0,C 180,E1 -26707.922,E2 -26707.922} C_VEL
LIN {X 0,Y 100.253,Z 318.742,A -85,B 0,C 180,E1 -26713.716,E2 -26713.716} C_VEL
LIN {X 0,Y 99.052,Z 320.48,A -85,B 0,C 180,E1 -26717.711,E2 -26717.711} C_VEL
LIN {X 0,Y 98.293,Z 321.724,A -85,B 0,C 180,E1 -26721.78,E2 -26721.78} C_VEL
LIN {X 0,Y 97.954,Z 322.496,A -85,B 0,C 180,E1 -26725.887,E2 -26725.887} C_VEL
LIN {X 0,Y 98.005,Z 322.79,A -85,B 0,C 180,E1 -26730.001,E2 -26730.001} C_VEL
LIN {X 0,Y 97.954,Z 322.483,A -85,B 0,C 180,E1 -26734.115,E2 -26734.115} C_VEL
LIN {X 0,Y 98.291,Z 321.685,A -85,B 0,C 180,E1 -26738.223,E2 -26738.223} C_VEL
LIN {X 0,Y 99.035,Z 320.414,A -85,B 0,C 180,E1 -26742.293,E2 -26742.293} C_VEL
LIN {X 0,Y 100.96,Z 317.491,A -85,B 0,C 180,E1 -26748.256,E2 -26748.256} C_VEL
LIN {X 0,Y 102.824,Z 314.828,A -85,B 0,C 180,E1 -26752.082,E2 -26752.082} C_VEL
LIN {X 0,Y 106.336,Z 309.63,A -85,B 0,C 180,E1 -26757.559,E2 -26757.559} C_VEL
LIN {X 0,Y 110.871,Z 302.776,A -85,B 0,C 180,E1 -26762.603,E2 -26762.603} C_VEL
LIN {X 0,Y 115.18,Z 295.291,A -85,B 0,C 180,E1 -26766.508,E2 -26766.508} C_VEL
LIN {X 0,Y 119.072,Z 287.911,A -85,B 0,C 180,E1 -26769.384,E2 -26769.384} C_VEL
LIN {X 0,Y 122.317,Z 280.838,A -85,B 0,C 180,E1 -26771.535,E2 -26771.535} C_VEL
LIN {X 0,Y 125.35,Z 273.139,A -85,B 0,C 180,E1 -26773.38,E2 -26773.38} C_VEL
LIN {X 0,Y 128.066,Z 264.737,A -85,B 0,C 180,E1 -26774.956,E2 -26774.956} C_VEL
LIN {X 0,Y 130.496,Z 255.837,A -85,B 0,C 180,E1 -26776.152,E2 -26776.152} C_VEL
LIN {X 0,Y 132.582,Z 245.46,A -85,B 0,C 180,E1 -26777.136,E2 -26777.136} C_VEL
LIN {X 0,Y 134.025,Z 231.734,A -85,B 0,C 180,E1 -26777.931,E2 -26777.931} C_VEL
LIN {X 0,Y 134.545,Z 223.539,A -85,B 0,C 180,E1 -26778.326,E2 -26778.326} C_VEL
LIN {X 0,Y 130.496,Z 212.244,A -85,B 0,C 180,E1 -26781.314,E2 -26781.314} C_VEL
LIN {X 0,Y 128.681,Z 208.43,A -85,B 0,C 180,E1 -26782.671,E2 -26782.671} C_VEL
LIN {X 0,Y 124.704,Z 201.734,A -85,B 0,C 180,E1 -26785.787,E2 -26785.787} C_VEL
LIN {X 0,Y 120.785,Z 195.815,A -85,B 0,C 180,E1 -26789.274,E2 -26789.274} C_VEL
LIN {X 0,Y 118.07,Z 191.878,A -85,B 0,C 180,E1 -26792.047,E2 -26792.047} C_VEL
LIN {X 0,Y 115.692,Z 188.612,A -85,B 0,C 180,E1 -26794.8,E2 -26794.8} C_VEL
LIN {X 0,Y 114.583,Z 187.401,A -85,B 0,C 180,E1 -26796.178,E2 -26796.178} C_VEL
LIN {X 0,Y 112.813,Z 187.203,A -85,B 0,C 180,E1 -26798.322,E2 -26798.322} C_VEL
LIN {X 0,Y 109.041,Z 188.658,A -85,B 0,C 180,E1 -26803.641,E2 -26803.641} C_VEL
LIN {X 0,Y 108.322,Z 188.396,A -85,B 0,C 180,E1 -26805.041,E2 -26805.041} C_VEL
LIN {X 0,Y 106.507,Z 185.557,A -85,B 0,C 180,E1 -26810.266,E2 -26810.266} C_VEL
LIN {X 0,Y 105.964,Z 184.089,A -85,B 0,C 180,E1 -26812.857,E2 -26812.857} C_VEL
LIN {X 0,Y 105.211,Z 183.244,A -85,B 0,C 180,E1 -26820,E2 -26820} C_VEL
LIN {X 0,Y 106.155,Z 184.345,A -85,B 0,C 180,E1 -26828.328,E2 -26828.328} C_VEL
LIN {X 0,Y 107.658,Z 187.68,A -85,B 0,C 180,E1 -26833.689,E2 -26833.689} C_VEL
LIN {X 0,Y 109.882,Z 189.67,A -85,B 0,C 180,E1 -26838.289,E2 -26838.289} C_VEL
LIN {X 0,Y 111.957,Z 193.116,A -85,B 0,C 180,E1 -26841.884,E2 -26841.884} C_VEL
LIN {X 0,Y 113.576,Z 194.888,A -85,B 0,C 180,E1 -26844.121,E2 -26844.121} C_VEL
LIN {X 0,Y 116.71,Z 199.467,A -85,B 0,C 180,E1 -26847.972,E2 -26847.972} C_VEL
LIN {X 0,Y 119.788,Z 204.249,A -85,B 0,C 180,E1 -26851.193,E2 -26851.193} C_VEL
LIN {X 0,Y 123.419,Z 210.203,A -85,B 0,C 180,E1 -26854.496,E2 -26854.496} C_VEL
LIN {X 0,Y 127.83,Z 218.414,A -85,B 0,C 180,E1 -26858.033,E2 -26858.033} C_VEL
LIN {X 0,Y 129.992,Z 223.115,A -85,B 0,C 180,E1 -26859.643,E2 -26859.643} C_VEL
LIN {X 0,Y 128.429,Z 239.936,A -85,B 0,C 180,E1 -26860.491,E2 -26860.491} C_VEL
LIN {X 0,Y 126.431,Z 250.903,A -85,B 0,C 180,E1 -26861.501,E2 -26861.501} C_VEL
LIN {X 0,Y 124.233,Z 259.556,A -85,B 0,C 180,E1 -26862.656,E2 -26862.656} C_VEL
LIN {X 0,Y 121.396,Z 268.362,A -85,B 0,C 180,E1 -26864.247,E2 -26864.247} C_VEL
LIN {X 0,Y 118.05,Z 276.708,A -85,B 0,C 180,E1 -26866.204,E2 -26866.204} C_VEL
LIN {X 0,Y 114.341,Z 284.612,A -85,B 0,C 180,E1 -26868.642,E2 -26868.642} C_VEL
LIN {X 0,Y 110.316,Z 291.984,A -85,B 0,C 180,E1 -26871.599,E2 -26871.599} C_VEL
LIN {X 0,Y 105.698,Z 299.453,A -85,B 0,C 180,E1 -26875.584,E2 -26875.584} C_VEL
LIN {X 0,Y 100.879,Z 306.292,A -85,B 0,C 180,E1 -26880.811,E2 -26880.811} C_VEL
LIN {X 0,Y 96.954,Z 311.464,A -85,B 0,C 180,E1 -26886.503,E2 -26886.503} C_VEL
LIN {X 0,Y 94.888,Z 314.114,A -85,B 0,C 180,E1 -26890.53,E2 -26890.53} C_VEL
LIN {X 0,Y 92.603,Z 317.015,A -85,B 0,C 180,E1 -26896.838,E2 -26896.838} C_VEL
LIN {X 0,Y 91.681,Z 318.276,A -85,B 0,C 180,E1 -26901.18,E2 -26901.18} C_VEL
LIN {X 0,Y 91.082,Z 319.069,A -85,B 0,C 180,E1 -26905.574,E2 -26905.574} C_VEL
LIN {X 0,Y 90.942,Z 319.371,A -85,B 0,C 180,E1 -26909.999,E2 -26909.999} C_VEL
LIN {X 0,Y 91.079,Z 319.089,A -85,B 0,C 180,E1 -26914.424,E2 -26914.424} C_VEL
LIN {X 0,Y 91.623,Z 318.336,A -85,B 0,C 180,E1 -26918.824,E2 -26918.824} C_VEL
LIN {X 0,Y 92.57,Z 317.115,A -85,B 0,C 180,E1 -26923.164,E2 -26923.164} C_VEL
LIN {X 0,Y 94.853,Z 314.256,A -85,B 0,C 180,E1 -26929.475,E2 -26929.475} C_VEL
LIN {X 0,Y 96.905,Z 311.651,A -85,B 0,C 180,E1 -26933.507,E2 -26933.507} C_VEL
LIN {X 0,Y 100.831,Z 306.529,A -85,B 0,C 180,E1 -26939.202,E2 -26939.202} C_VEL
LIN {X 0,Y 104.788,Z 301.016,A -85,B 0,C 180,E1 -26943.593,E2 -26943.593} C_VEL
LIN {X 0,Y 109.285,Z 294.082,A -85,B 0,C 180,E1 -26947.656,E2 -26947.656} C_VEL
LIN {X 0,Y 113.766,Z 286.12,A -85,B 0,C 180,E1 -26951.022,E2 -26951.022} C_VEL
LIN {X 0,Y 117.53,Z 278.527,A -85,B 0,C 180,E1 -26953.445,E2 -26953.445} C_VEL
LIN {X 0,Y 120.866,Z 270.446,A -85,B 0,C 180,E1 -26955.468,E2 -26955.468} C_VEL
LIN {X 0,Y 123.805,Z 261.877,A -85,B 0,C 180,E1 -26957.103,E2 -26957.103} C_VEL
LIN {X 0,Y 126.229,Z 252.828,A -85,B 0,C 180,E1 -26958.412,E2 -26958.412} C_VEL
LIN {X 0,Y 128.323,Z 242.214,A -85,B 0,C 180,E1 -26959.487,E2 -26959.487} C_VEL
LIN {X 0,Y 129.811,Z 228.243,A -85,B 0,C 180,E1 -26960.309,E2 -26960.309} C_VEL
LIN {X 0,Y 130.191,Z 223.267,A -85,B 0,C 180,E1 -26960.529,E2 -26960.529} C_VEL
LIN {X 0,Y 125.798,Z 214.263,A -85,B 0,C 180,E1 -26963.883,E2 -26963.883} C_VEL
LIN {X 0,Y 120.942,Z 205.842,A -85,B 0,C 180,E1 -26968.098,E2 -26968.098} C_VEL
LIN {X 0,Y 117.796,Z 201.087,A -85,B 0,C 180,E1 -26971.247,E2 -26971.247} C_VEL
LIN {X 0,Y 115.798,Z 198.052,A -85,B 0,C 180,E1 -26973.524,E2 -26973.524} C_VEL
LIN {X 0,Y 113.042,Z 194.05,A -85,B 0,C 180,E1 -26977.134,E2 -26977.134} C_VEL
LIN {X 0,Y 110.598,Z 191.045,A -85,B 0,C 180,E1 -26980.952,E2 -26980.952} C_VEL
LIN {X 0,Y 109.692,Z 189.285,A -85,B 0,C 180,E1 -26982.763,E2 -26982.763} C_VEL
LIN {X 0,Y 107.369,Z 187.166,A -85,B 0,C 180,E1 -26988.054,E2 -26988.054} C_VEL
LIN {X 0,Y 106.153,Z 184.264,A -85,B 0,C 180,E1 -26993.252,E2 -26993.252} C_VEL
LIN {X 0,Y 105.544,Z 183.42,A -85,B 0,C 180,E1 -27000,E2 -27000} C_VEL
LIN {X 0,Y 106.191,Z 184.333,A -85,B 0,C 180,E1 -27006.747,E2 -27006.747} C_VEL
LIN {X 0,Y 108.347,Z 188.341,A -85,B 0,C 180,E1 -27014.302,E2 -27014.302} C_VEL
LIN {X 0,Y 109.962,Z 189.637,A -85,B 0,C 180,E1 -27017.553,E2 -27017.553} C_VEL
LIN {X 0,Y 111.98,Z 193.062,A -85,B 0,C 180,E1 -27021.154,E2 -27021.154} C_VEL
LIN {X 0,Y 113.703,Z 194.893,A -85,B 0,C 180,E1 -27023.567,E2 -27023.567} C_VEL
LIN {X 0,Y 116.975,Z 199.77,A -85,B 0,C 180,E1 -27027.629,E2 -27027.629} C_VEL
LIN {X 0,Y 120.315,Z 204.927,A -85,B 0,C 180,E1 -27031.104,E2 -27031.104} C_VEL
LIN {X 0,Y 124.683,Z 212.257,A -85,B 0,C 180,E1 -27035,E2 -27035} C_VEL
LIN {X 0,Y 126.749,Z 216.608,A -85,B 0,C 180,E1 -27036.712,E2 -27036.712} C_VEL
LIN {X 0,Y 129.951,Z 225.874,A -85,B 0,C 180,E1 -27039.355,E2 -27039.355} C_VEL
LIN {X 0,Y 128.428,Z 243.054,A -85,B 0,C 180,E1 -27040.26,E2 -27040.26} C_VEL
LIN {X 0,Y 126.519,Z 253.216,A -85,B 0,C 180,E1 -27041.128,E2 -27041.128} C_VEL
LIN {X 0,Y 123.788,Z 263.352,A -85,B 0,C 180,E1 -27042.434,E2 -27042.434} C_VEL
LIN {X 0,Y 120.833,Z 272.003,A -85,B 0,C 180,E1 -27043.966,E2 -27043.966} C_VEL
LIN {X 0,Y 117.873,Z 279.363,A -85,B 0,C 180,E1 -27045.682,E2 -27045.682} C_VEL
LIN {X 0,Y 114.219,Z 287.09,A -85,B 0,C 180,E1 -27048,E2 -27048} C_VEL
LIN {X 0,Y 110.567,Z 293.734,A -85,B 0,C 180,E1 -27050.534,E2 -27050.534} C_VEL
LIN {X 0,Y 106.724,Z 300.045,A -85,B 0,C 180,E1 -27053.655,E2 -27053.655} C_VEL
LIN {X 0,Y 103.236,Z 305.289,A -85,B 0,C 180,E1 -27057.003,E2 -27057.003} C_VEL
LIN {X 0,Y 100.107,Z 309.661,A -85,B 0,C 180,E1 -27060.566,E2 -27060.566} C_VEL
LIN {X 0,Y 96.266,Z 314.823,A -85,B 0,C 180,E1 -27066.327,E2 -27066.327} C_VEL
LIN {X 0,Y 93.444,Z 318.614,A -85,B 0,C 180,E1 -27072.493,E2 -27072.493} C_VEL
LIN {X 0,Y 92.12,Z 320.352,A -85,B 0,C 180,E1 -27076.77,E2 -27076.77} C_VEL
LIN {X 0,Y 91.264,Z 321.596,A -85,B 0,C 180,E1 -27081.141,E2 -27081.141} C_VEL
LIN {X 0,Y 90.885,Z 322.368,A -85,B 0,C 180,E1 -27085.566,E2 -27085.566} C_VEL
LIN {X 0,Y 90.912,Z 322.661,A -85,B 0,C 180,E1 -27090.001,E2 -27090.001} C_VEL
LIN {X 0,Y 90.885,Z 322.355,A -85,B 0,C 180,E1 -27094.436,E2 -27094.436} C_VEL
LIN {X 0,Y 91.261,Z 321.556,A -85,B 0,C 180,E1 -27098.861,E2 -27098.861} C_VEL
LIN {X 0,Y 92.102,Z 320.284,A -85,B 0,C 180,E1 -27103.235,E2 -27103.235} C_VEL
LIN {X 0,Y 94.228,Z 317.361,A -85,B 0,C 180,E1 -27109.612,E2 -27109.612} C_VEL
LIN {X 0,Y 96.255,Z 314.698,A -85,B 0,C 180,E1 -27113.678,E2 -27113.678} C_VEL
LIN {X 0,Y 100.095,Z 309.5,A -85,B 0,C 180,E1 -27119.44,E2 -27119.44} C_VEL
LIN {X 0,Y 104.964,Z 302.646,A -85,B 0,C 180,E1 -27124.69,E2 -27124.69} C_VEL
LIN {X 0,Y 109.555,Z 295.16,A -85,B 0,C 180,E1 -27128.717,E2 -27128.717} C_VEL
LIN {X 0,Y 113.666,Z 287.779,A -85,B 0,C 180,E1 -27131.659,E2 -27131.659} C_VEL
LIN {X 0,Y 117.128,Z 280.637,A -85,B 0,C 180,E1 -27133.858,E2 -27133.858} C_VEL
LIN {X 0,Y 120.289,Z 273.006,A -85,B 0,C 180,E1 -27135.703,E2 -27135.703} C_VEL
LIN {X 0,Y 123.141,Z 264.602,A -85,B 0,C 180,E1 -27137.292,E2 -27137.292} C_VEL
LIN {X 0,Y 125.548,Z 256.28,A -85,B 0,C 180,E1 -27138.411,E2 -27138.411} C_VEL
LIN {X 0,Y 127.566,Z 246.814,A -85,B 0,C 180,E1 -27139.35,E2 -27139.35} C_VEL
LIN {X 0,Y 129.059,Z 235.51,A -85,B 0,C 180,E1 -27140.091,E2 -27140.091} C_VEL
LIN {X 0,Y 129.744,Z 225.647,A -85,B 0,C 180,E1 -27140.574,E2 -27140.574} C_VEL
LIN {X 0,Y 126.274,Z 215.673,A -85,B 0,C 180,E1 -27143.438,E2 -27143.438} C_VEL
LIN {X 0,Y 123.395,Z 210.15,A -85,B 0,C 180,E1 -27145.825,E2 -27145.825} C_VEL
LIN {X 0,Y 119.98,Z 204.529,A -85,B 0,C 180,E1 -27148.922,E2 -27148.922} C_VEL
LIN {X 0,Y 115.885,Z 198.18,A -85,B 0,C 180,E1 -27153.283,E2 -27153.283} C_VEL
LIN {X 0,Y 113.092,Z 194.12,A -85,B 0,C 180,E1 -27156.857,E2 -27156.857} C_VEL
LIN {X 0,Y 110.592,Z 191.173,A -85,B 0,C 180,E1 -27160.632,E2 -27160.632} C_VEL
LIN {X 0,Y 109.551,Z 189.221,A -85,B 0,C 180,E1 -27162.642,E2 -27162.642} C_VEL
LIN {X 0,Y 108.322,Z 188.396,A -85,B 0,C 180,E1 -27165.041,E2 -27165.041} C_VEL
LIN {X 0,Y 107.012,Z 187.752,A -85,B 0,C 180,E1 -27168.108,E2 -27168.108} C_VEL
LIN {X 0,Y 105.31,Z 188.405,A -85,B 0,C 180,E1 -27173.386,E2 -27173.386} C_VEL
LIN {X 0,Y 104.381,Z 190.5,A -85,B 0,C 180,E1 -27182.114,E2 -27182.114} C_VEL
LIN {X 0,Y 105.083,Z 191.213,A -85,B 0,C 180,E1 -27187.446,E2 -27187.446} C_VEL
LIN {X 0,Y 106.373,Z 194.431,A -85,B 0,C 180,E1 -27192.687,E2 -27192.687} C_VEL
LIN {X 0,Y 108.361,Z 196.431,A -85,B 0,C 180,E1 -27197.213,E2 -27197.213} C_VEL
LIN {X 0,Y 110.601,Z 200.073,A -85,B 0,C 180,E1 -27201.309,E2 -27201.309} C_VEL
LIN {X 0,Y 111.679,Z 201.377,A -85,B 0,C 180,E1 -27202.909,E2 -27202.909} C_VEL
LIN {X 0,Y 114.498,Z 205.723,A -85,B 0,C 180,E1 -27206.67,E2 -27206.67} C_VEL
LIN {X 0,Y 117.29,Z 210.31,A -85,B 0,C 180,E1 -27209.845,E2 -27209.845} C_VEL
LIN {X 0,Y 121.511,Z 217.714,A -85,B 0,C 180,E1 -27213.947,E2 -27213.947} C_VEL
LIN {X 0,Y 125.371,Z 225.754,A -85,B 0,C 180,E1 -27217.252,E2 -27217.252} C_VEL
LIN {X 0,Y 123.771,Z 241.241,A -85,B 0,C 180,E1 -27218.082,E2 -27218.082} C_VEL
LIN {X 0,Y 121.572,Z 252.182,A -85,B 0,C 180,E1 -27219.154,E2 -27219.154} C_VEL
LIN {X 0,Y 119.169,Z 260.834,A -85,B 0,C 180,E1 -27220.343,E2 -27220.343} C_VEL
LIN {X 0,Y 116.625,Z 268.314,A -85,B 0,C 180,E1 -27221.707,E2 -27221.707} C_VEL
LIN {X 0,Y 113.029,Z 276.841,A -85,B 0,C 180,E1 -27223.71,E2 -27223.71} C_VEL
LIN {X 0,Y 109.125,Z 284.743,A -85,B 0,C 180,E1 -27226.184,E2 -27226.184} C_VEL
LIN {X 0,Y 104.85,Z 292.115,A -85,B 0,C 180,E1 -27229.19,E2 -27229.19} C_VEL
LIN {X 0,Y 99.909,Z 299.584,A -85,B 0,C 180,E1 -27233.277,E2 -27233.277} C_VEL
LIN {X 0,Y 94.737,Z 306.422,A -85,B 0,C 180,E1 -27238.714,E2 -27238.714} C_VEL
LIN {X 0,Y 90.489,Z 311.594,A -85,B 0,C 180,E1 -27244.711,E2 -27244.711} C_VEL
LIN {X 0,Y 88.228,Z 314.243,A -85,B 0,C 180,E1 -27248.993,E2 -27248.993} C_VEL
LIN {X 0,Y 85.695,Z 317.144,A -85,B 0,C 180,E1 -27255.756,E2 -27255.756} C_VEL
LIN {X 0,Y 84.672,Z 318.405,A -85,B 0,C 180,E1 -27260.443,E2 -27260.443} C_VEL
LIN {X 0,Y 84.014,Z 319.198,A -85,B 0,C 180,E1 -27265.2,E2 -27265.2} C_VEL
LIN {X 0,Y 83.843,Z 319.499,A -85,B 0,C 180,E1 -27269.999,E2 -27269.999} C_VEL
LIN {X 0,Y 84.01,Z 319.217,A -85,B 0,C 180,E1 -27274.798,E2 -27274.798} C_VEL
LIN {X 0,Y 84.628,Z 318.464,A -85,B 0,C 180,E1 -27279.559,E2 -27279.559} C_VEL
LIN {X 0,Y 85.668,Z 317.243,A -85,B 0,C 180,E1 -27284.246,E2 -27284.246} C_VEL
LIN {X 0,Y 88.194,Z 314.383,A -85,B 0,C 180,E1 -27291.013,E2 -27291.013} C_VEL
LIN {X 0,Y 90.444,Z 311.778,A -85,B 0,C 180,E1 -27295.3,E2 -27295.3} C_VEL
LIN {X 0,Y 94.69,Z 306.656,A -85,B 0,C 180,E1 -27301.301,E2 -27301.301} C_VEL
LIN {X 0,Y 98.956,Z 301.143,A -85,B 0,C 180,E1 -27305.867,E2 -27305.867} C_VEL
LIN {X 0,Y 103.753,Z 294.208,A -85,B 0,C 180,E1 -27310.052,E2 -27310.052} C_VEL
LIN {X 0,Y 108.523,Z 286.245,A -85,B 0,C 180,E1 -27313.477,E2 -27313.477} C_VEL
LIN {X 0,Y 112.484,Z 278.652,A -85,B 0,C 180,E1 -27315.931,E2 -27315.931} C_VEL
LIN {X 0,Y 116.029,Z 270.508,A -85,B 0,C 180,E1 -27317.978,E2 -27317.978} C_VEL
LIN {X 0,Y 118.761,Z 262.994,A -85,B 0,C 180,E1 -27319.442,E2 -27319.442} C_VEL
LIN {X 0,Y 121.464,Z 253.698,A -85,B 0,C 180,E1 -27320.808,E2 -27320.808} C_VEL
LIN {X 0,Y 123.469,Z 244.283,A -85,B 0,C 180,E1 -27321.811,E2 -27321.811} C_VEL
LIN {X 0,Y 124.832,Z 234.422,A -85,B 0,C 180,E1 -27322.51,E2 -27322.51} C_VEL
LIN {X 0,Y 125.561,Z 225.835,A -85,B 0,C 180,E1 -27322.94,E2 -27322.94} C_VEL
LIN {X 0,Y 121.281,Z 217.143,A -85,B 0,C 180,E1 -27326.627,E2 -27326.627} C_VEL
LIN {X 0,Y 117.348,Z 210.231,A -85,B 0,C 180,E1 -27330.513,E2 -27330.513} C_VEL
LIN {X 0,Y 113.817,Z 204.475,A -85,B 0,C 180,E1 -27334.665,E2 -27334.665} C_VEL
LIN {X 0,Y 111.258,Z 200.589,A -85,B 0,C 180,E1 -27338.282,E2 -27338.282} C_VEL
LIN {X 0,Y 108.877,Z 197.36,A -85,B 0,C 180,E1 -27342.387,E2 -27342.387} C_VEL
LIN {X 0,Y 108.15,Z 196.018,A -85,B 0,C 180,E1 -27343.967,E2 -27343.967} C_VEL
LIN {X 0,Y 106.094,Z 193.777,A -85,B 0,C 180,E1 -27349.262,E2 -27349.262} C_VEL
LIN {X 0,Y 105.109,Z 191.125,A -85,B 0,C 180,E1 -27354.243,E2 -27354.243} C_VEL
LIN {X 0,Y 104.678,Z 190.475,A -85,B 0,C 180,E1 -27360,E2 -27360} C_VEL
LIN {X 0,Y 105.263,Z 191.469,A -85,B 0,C 180,E1 -27366.542,E2 -27366.542} C_VEL
LIN {X 0,Y 107.021,Z 195.093,A -85,B 0,C 180,E1 -27373.287,E2 -27373.287} C_VEL
LIN {X 0,Y 108.465,Z 196.368,A -85,B 0,C 180,E1 -27376.477,E2 -27376.477} C_VEL
LIN {X 0,Y 110.548,Z 199.894,A -85,B 0,C 180,E1 -27380.433,E2 -27380.433} C_VEL
LIN {X 0,Y 111.78,Z 201.348,A -85,B 0,C 180,E1 -27382.299,E2 -27382.299} C_VEL
LIN {X 0,Y 114.778,Z 206.027,A -85,B 0,C 180,E1 -27386.339,E2 -27386.339} C_VEL
LIN {X 0,Y 117.689,Z 210.786,A -85,B 0,C 180,E1 -27389.638,E2 -27389.638} C_VEL
LIN {X 0,Y 121.567,Z 217.641,A -85,B 0,C 180,E1 -27393.421,E2 -27393.421} C_VEL
LIN {X 0,Y 123.384,Z 221.881,A -85,B 0,C 180,E1 -27395.096,E2 -27395.096} C_VEL
LIN {X 0,Y 125.37,Z 227.988,A -85,B 0,C 180,E1 -27396.935,E2 -27396.935} C_VEL
LIN {X 0,Y 123.931,Z 243.092,A -85,B 0,C 180,E1 -27397.762,E2 -27397.762} C_VEL
LIN {X 0,Y 121.663,Z 254.211,A -85,B 0,C 180,E1 -27398.74,E2 -27398.74} C_VEL
LIN {X 0,Y 119.109,Z 263.23,A -85,B 0,C 180,E1 -27399.911,E2 -27399.911} C_VEL
LIN {X 0,Y 116.018,Z 271.879,A -85,B 0,C 180,E1 -27401.443,E2 -27401.443} C_VEL
LIN {X 0,Y 112.445,Z 280.213,A -85,B 0,C 180,E1 -27403.433,E2 -27403.433} C_VEL
LIN {X 0,Y 108.505,Z 287.987,A -85,B 0,C 180,E1 -27405.871,E2 -27405.871} C_VEL
LIN {X 0,Y 104.112,Z 295.315,A -85,B 0,C 180,E1 -27408.841,E2 -27408.841} C_VEL
LIN {X 0,Y 99.22,Z 302.751,A -85,B 0,C 180,E1 -27412.983,E2 -27412.983} C_VEL
LIN {X 0,Y 94.806,Z 308.576,A -85,B 0,C 180,E1 -27417.491,E2 -27417.491} C_VEL
LIN {X 0,Y 91.032,Z 313.172,A -85,B 0,C 180,E1 -27422.406,E2 -27422.406} C_VEL
LIN {X 0,Y 88.643,Z 316.163,A -85,B 0,C 180,E1 -27426.647,E2 -27426.647} C_VEL
LIN {X 0,Y 86.695,Z 318.486,A -85,B 0,C 180,E1 -27431.08,E2 -27431.08} C_VEL
LIN {X 0,Y 85.226,Z 320.224,A -85,B 0,C 180,E1 -27435.678,E2 -27435.678} C_VEL
LIN {X 0,Y 84.242,Z 321.468,A -85,B 0,C 180,E1 -27440.396,E2 -27440.396} C_VEL
LIN {X 0,Y 83.804,Z 322.24,A -85,B 0,C 180,E1 -27445.191,E2 -27445.191} C_VEL
LIN {X 0,Y 83.811,Z 322.533,A -85,B 0,C 180,E1 -27450.001,E2 -27450.001} C_VEL
LIN {X 0,Y 83.804,Z 322.226,A -85,B 0,C 180,E1 -27454.812,E2 -27454.812} C_VEL
LIN {X 0,Y 84.239,Z 321.427,A -85,B 0,C 180,E1 -27459.606,E2 -27459.606} C_VEL
LIN {X 0,Y 85.208,Z 320.155,A -85,B 0,C 180,E1 -27464.327,E2 -27464.327} C_VEL
LIN {X 0,Y 87.566,Z 317.232,A -85,B 0,C 180,E1 -27471.173,E2 -27471.173} C_VEL
LIN {X 0,Y 89.778,Z 314.568,A -85,B 0,C 180,E1 -27475.504,E2 -27475.504} C_VEL
LIN {X 0,Y 93.981,Z 309.37,A -85,B 0,C 180,E1 -27481.566,E2 -27481.566} C_VEL
LIN {X 0,Y 99.214,Z 302.515,A -85,B 0,C 180,E1 -27487.023,E2 -27487.023} C_VEL
LIN {X 0,Y 104.115,Z 295.029,A -85,B 0,C 180,E1 -27491.16,E2 -27491.16} C_VEL
LIN {X 0,Y 108.464,Z 287.647,A -85,B 0,C 180,E1 -27494.152,E2 -27494.152} C_VEL
LIN {X 0,Y 112.365,Z 279.959,A -85,B 0,C 180,E1 -27496.528,E2 -27496.528} C_VEL
LIN {X 0,Y 116.052,Z 271.372,A -85,B 0,C 180,E1 -27498.541,E2 -27498.541} C_VEL
LIN {X 0,Y 119.748,Z 260.554,A -85,B 0,C 180,E1 -27500.411,E2 -27500.411} C_VEL
LIN {X 0,Y 122.443,Z 249.767,A -85,B 0,C 180,E1 -27501.608,E2 -27501.608} C_VEL
LIN {X 0,Y 123.997,Z 240.607,A -85,B 0,C 180,E1 -27502.301,E2 -27502.301} C_VEL
LIN {X 0,Y 125.198,Z 227.923,A -85,B 0,C 180,E1 -27502.95,E2 -27502.95} C_VEL
LIN {X 0,Y 122.208,Z 219.155,A -85,B 0,C 180,E1 -27505.721,E2 -27505.721} C_VEL
LIN {X 0,Y 118.193,Z 211.706,A -85,B 0,C 180,E1 -27509.533,E2 -27509.533} C_VEL
LIN {X 0,Y 115.064,Z 206.686,A -85,B 0,C 180,E1 -27512.942,E2 -27512.942} C_VEL
LIN {X 0,Y 113.363,Z 203.97,A -85,B 0,C 180,E1 -27515.059,E2 -27515.059} C_VEL
LIN {X 0,Y 111.148,Z 200.544,A -85,B 0,C 180,E1 -27518.193,E2 -27518.193} C_VEL
LIN {X 0,Y 108.797,Z 197.377,A -85,B 0,C 180,E1 -27522.155,E2 -27522.155} C_VEL
LIN {X 0,Y 108.181,Z 196.042,A -85,B 0,C 180,E1 -27523.488,E2 -27523.488} C_VEL
LIN {X 0,Y 105.994,Z 193.835,A -85,B 0,C 180,E1 -27528.769,E2 -27528.769} C_VEL
LIN {X 0,Y 105.001,Z 191.097,A -85,B 0,C 180,E1 -27533.274,E2 -27533.274} C_VEL
LIN {X 0,Y 104.344,Z 190.305,A -85,B 0,C 180,E1 -27540,E2 -27540} C_VEL
LIN {X 0,Y 104.381,Z 190.5,A -85,B 0,C 180,E1 -27542.114,E2 -27542.114} C_VEL
LIN {X 0,Y 104.446,Z 191.578,A -85,B 0,C 180,E1 -27544.183,E2 -27544.183} C_VEL
LIN {X 0,Y 104.493,Z 195.478,A -85,B 0,C 180,E1 -27547.174,E2 -27547.174} C_VEL
LIN {X 0,Y 104.765,Z 199.755,A -85,B 0,C 180,E1 -27550.118,E2 -27550.118} C_VEL
LIN {X 0,Y 105.274,Z 201.381,A -85,B 0,C 180,E1 -27552.123,E2 -27552.123} C_VEL
LIN {X 0,Y 106.884,Z 203.146,A -85,B 0,C 180,E1 -27556.105,E2 -27556.105} C_VEL
LIN {X 0,Y 109.123,Z 206.852,A -85,B 0,C 180,E1 -27560.5,E2 -27560.5} C_VEL
LIN {X 0,Y 110.345,Z 208.74,A -85,B 0,C 180,E1 -27562.467,E2 -27562.467} C_VEL
LIN {X 0,Y 112.309,Z 211.898,A -85,B 0,C 180,E1 -27565.264,E2 -27565.264} C_VEL
LIN {X 0,Y 115.64,Z 217.703,A -85,B 0,C 180,E1 -27569.315,E2 -27569.315} C_VEL
LIN {X 0,Y 119.634,Z 225.581,A -85,B 0,C 180,E1 -27573.431,E2 -27573.431} C_VEL
LIN {X 0,Y 120.965,Z 228.565,A -85,B 0,C 180,E1 -27574.687,E2 -27574.687} C_VEL
LIN {X 0,Y 119.276,Z 242.669,A -85,B 0,C 180,E1 -27575.511,E2 -27575.511} C_VEL
LIN {X 0,Y 117.249,Z 252.229,A -85,B 0,C 180,E1 -27576.455,E2 -27576.455} C_VEL
LIN {X 0,Y 114.655,Z 261.125,A -85,B 0,C 180,E1 -27577.67,E2 -27577.67} C_VEL
LIN {X 0,Y 111.618,Z 269.445,A -85,B 0,C 180,E1 -27579.213,E2 -27579.213} C_VEL
LIN {X 0,Y 108.255,Z 276.973,A -85,B 0,C 180,E1 -27580.999,E2 -27580.999} C_VEL
LIN {X 0,Y 104.12,Z 284.875,A -85,B 0,C 180,E1 -27583.479,E2 -27583.479} C_VEL
LIN {X 0,Y 99.593,Z 292.246,A -85,B 0,C 180,E1 -27586.524,E2 -27586.524} C_VEL
LIN {X 0,Y 94.31,Z 299.715,A -85,B 0,C 180,E1 -27590.696,E2 -27590.696} C_VEL
LIN {X 0,Y 88.741,Z 306.553,A -85,B 0,C 180,E1 -27596.331,E2 -27596.331} C_VEL
LIN {X 0,Y 84.132,Z 311.724,A -85,B 0,C 180,E1 -27602.647,E2 -27602.647} C_VEL
LIN {X 0,Y 81.647,Z 314.372,A -85,B 0,C 180,E1 -27607.209,E2 -27607.209} C_VEL
LIN {X 0,Y 78.835,Z 317.273,A -85,B 0,C 180,E1 -27614.487,E2 -27614.487} C_VEL
LIN {X 0,Y 77.695,Z 318.533,A -85,B 0,C 180,E1 -27619.576,E2 -27619.576} C_VEL
LIN {X 0,Y 76.941,Z 319.326,A -85,B 0,C 180,E1 -27624.758,E2 -27624.758} C_VEL
LIN {X 0,Y 76.759,Z 319.627,A -85,B 0,C 180,E1 -27629.999,E2 -27629.999} C_VEL
LIN {X 0,Y 76.938,Z 319.346,A -85,B 0,C 180,E1 -27635.24,E2 -27635.24} C_VEL
LIN {X 0,Y 77.627,Z 318.592,A -85,B 0,C 180,E1 -27640.431,E2 -27640.431} C_VEL
LIN {X 0,Y 78.813,Z 317.371,A -85,B 0,C 180,E1 -27645.515,E2 -27645.515} C_VEL
LIN {X 0,Y 81.615,Z 314.51,A -85,B 0,C 180,E1 -27652.798,E2 -27652.798} C_VEL
LIN {X 0,Y 84.09,Z 311.905,A -85,B 0,C 180,E1 -27657.365,E2 -27657.365} C_VEL
LIN {X 0,Y 88.695,Z 306.783,A -85,B 0,C 180,E1 -27663.686,E2 -27663.686} C_VEL
LIN {X 0,Y 93.277,Z 301.27,A -85,B 0,C 180,E1 -27668.432,E2 -27668.432} C_VEL
LIN {X 0,Y 98.42,Z 294.334,A -85,B 0,C 180,E1 -27672.716,E2 -27672.716} C_VEL
LIN {X 0,Y 103.489,Z 286.37,A -85,B 0,C 180,E1 -27676.181,E2 -27676.181} C_VEL
LIN {X 0,Y 107.668,Z 278.776,A -85,B 0,C 180,E1 -27678.646,E2 -27678.646} C_VEL
LIN {X 0,Y 111.457,Z 270.5,A -85,B 0,C 180,E1 -27680.719,E2 -27680.719} C_VEL
LIN {X 0,Y 114.651,Z 262.059,A -85,B 0,C 180,E1 -27682.308,E2 -27682.308} C_VEL
LIN {X 0,Y 117.193,Z 253.43,A -85,B 0,C 180,E1 -27683.56,E2 -27683.56} C_VEL
LIN {X 0,Y 119.349,Z 243.663,A -85,B 0,C 180,E1 -27684.561,E2 -27684.561} C_VEL
LIN {X 0,Y 120.945,Z 232.244,A -85,B 0,C 180,E1 -27685.29,E2 -27685.29} C_VEL
LIN {X 0,Y 121.202,Z 228.805,A -85,B 0,C 180,E1 -27685.467,E2 -27685.467} C_VEL
LIN {X 0,Y 117.889,Z 221.857,A -85,B 0,C 180,E1 -27688.683,E2 -27688.683} C_VEL
LIN {X 0,Y 114.734,Z 215.956,A -85,B 0,C 180,E1 -27692.158,E2 -27692.158} C_VEL
LIN {X 0,Y 111.539,Z 210.44,A -85,B 0,C 180,E1 -27696.316,E2 -27696.316} C_VEL
LIN {X 0,Y 109.299,Z 206.869,A -85,B 0,C 180,E1 -27699.83,E2 -27699.83} C_VEL
LIN {X 0,Y 107.158,Z 203.509,A -85,B 0,C 180,E1 -27704.033,E2 -27704.033} C_VEL
LIN {X 0,Y 106.659,Z 202.73,A -85,B 0,C 180,E1 -27705.206,E2 -27705.206} C_VEL
LIN {X 0,Y 104.843,Z 200.355,A -85,B 0,C 180,E1 -27710.596,E2 -27710.596} C_VEL
LIN {X 0,Y 104.171,Z 198.122,A -85,B 0,C 180,E1 -27714.677,E2 -27714.677} C_VEL
LIN {X 0,Y 103.822,Z 197.596,A -85,B 0,C 180,E1 -27720.969,E2 -27720.969} C_VEL
LIN {X 0,Y 104.258,Z 198.402,A -85,B 0,C 180,E1 -27725.803,E2 -27725.803} C_VEL
LIN {X 0,Y 105.808,Z 201.929,A -85,B 0,C 180,E1 -27732.466,E2 -27732.466} C_VEL
LIN {X 0,Y 107.062,Z 203.262,A -85,B 0,C 180,E1 -27735.514,E2 -27735.514} C_VEL
LIN {X 0,Y 109.234,Z 206.846,A -85,B 0,C 180,E1 -27739.862,E2 -27739.862} C_VEL
LIN {X 0,Y 110.099,Z 208.077,A -85,B 0,C 180,E1 -27741.283,E2 -27741.283} C_VEL
LIN {X 0,Y 112.66,Z 212.32,A -85,B 0,C 180,E1 -27745.026,E2 -27745.026} C_VEL
LIN {X 0,Y 116.139,Z 218.442,A -85,B 0,C 180,E1 -27749.233,E2 -27749.233} C_VEL
LIN {X 0,Y 119.385,Z 224.998,A -85,B 0,C 180,E1 -27752.617,E2 -27752.617} C_VEL
LIN {X 0,Y 121.073,Z 230.328,A -85,B 0,C 180,E1 -27754.39,E2 -27754.39} C_VEL
LIN {X 0,Y 119.431,Z 244.733,A -85,B 0,C 180,E1 -27755.225,E2 -27755.225} C_VEL
LIN {X 0,Y 117.027,Z 255.249,A -85,B 0,C 180,E1 -27756.167,E2 -27756.167} C_VEL
LIN {X 0,Y 114.691,Z 263.107,A -85,B 0,C 180,E1 -27757.194,E2 -27757.194} C_VEL
LIN {X 0,Y 111.444,Z 271.755,A -85,B 0,C 180,E1 -27758.704,E2 -27758.704} C_VEL
LIN {X 0,Y 107.805,Z 279.846,A -85,B 0,C 180,E1 -27760.621,E2 -27760.621} C_VEL
LIN {X 0,Y 104.095,Z 286.839,A -85,B 0,C 180,E1 -27762.76,E2 -27762.76} C_VEL
LIN {X 0,Y 100.021,Z 293.483,A -85,B 0,C 180,E1 -27765.362,E2 -27765.362} C_VEL
LIN {X 0,Y 95.634,Z 299.792,A -85,B 0,C 180,E1 -27768.595,E2 -27768.595} C_VEL
LIN {X 0,Y 91.665,Z 305.036,A -85,B 0,C 180,E1 -27772.168,E2 -27772.168} C_VEL
LIN {X 0,Y 88.027,Z 309.407,A -85,B 0,C 180,E1 -27776.023,E2 -27776.023} C_VEL
LIN {X 0,Y 83.422,Z 314.568,A -85,B 0,C 180,E1 -27782.398,E2 -27782.398} C_VEL
LIN {X 0,Y 79.997,Z 318.358,A -85,B 0,C 180,E1 -27789.428,E2 -27789.428} C_VEL
LIN {X 0,Y 78.345,Z 320.096,A -85,B 0,C 180,E1 -27794.39,E2 -27794.39} C_VEL
LIN {X 0,Y 77.251,Z 321.34,A -85,B 0,C 180,E1 -27799.518,E2 -27799.518} C_VEL
LIN {X 0,Y 76.743,Z 322.112,A -85,B 0,C 180,E1 -27804.747,E2 -27804.747} C_VEL
LIN {X 0,Y 76.733,Z 322.405,A -85,B 0,C 180,E1 -27810.001,E2 -27810.001} C_VEL
LIN {X 0,Y 76.743,Z 322.098,A -85,B 0,C 180,E1 -27815.256,E2 -27815.256} C_VEL
LIN {X 0,Y 77.247,Z 321.298,A -85,B 0,C 180,E1 -27820.485,E2 -27820.485} C_VEL
LIN {X 0,Y 78.328,Z 320.026,A -85,B 0,C 180,E1 -27825.616,E2 -27825.616} C_VEL
LIN {X 0,Y 80.967,Z 317.102,A -85,B 0,C 180,E1 -27832.993,E2 -27832.993} C_VEL
LIN {X 0,Y 83.413,Z 314.438,A -85,B 0,C 180,E1 -27837.608,E2 -27837.608} C_VEL
LIN {X 0,Y 87.994,Z 309.24,A -85,B 0,C 180,E1 -27843.994,E2 -27843.994} C_VEL
LIN {X 0,Y 93.643,Z 302.385,A -85,B 0,C 180,E1 -27849.639,E2 -27849.639} C_VEL
LIN {X 0,Y 98.888,Z 294.898,A -85,B 0,C 180,E1 -27853.864,E2 -27853.864} C_VEL
LIN {X 0,Y 103.487,Z 287.516,A -85,B 0,C 180,E1 -27856.892,E2 -27856.892} C_VEL
LIN {X 0,Y 107.662,Z 279.706,A -85,B 0,C 180,E1 -27859.307,E2 -27859.307} C_VEL
LIN {X 0,Y 112.087,Z 269.735,A -85,B 0,C 180,E1 -27861.608,E2 -27861.608} C_VEL
LIN {X 0,Y 115.916,Z 258.506,A -85,B 0,C 180,E1 -27863.346,E2 -27863.346} C_VEL
LIN {X 0,Y 118.369,Z 248.715,A -85,B 0,C 180,E1 -27864.369,E2 -27864.369} C_VEL
LIN {X 0,Y 119.905,Z 239.54,A -85,B 0,C 180,E1 -27865.039,E2 -27865.039} C_VEL
LIN {X 0,Y 120.85,Z 230.133,A -85,B 0,C 180,E1 -27865.531,E2 -27865.531} C_VEL
LIN {X 0,Y 118.782,Z 223.867,A -85,B 0,C 180,E1 -27867.688,E2 -27867.688} C_VEL
LIN {X 0,Y 115.248,Z 217.012,A -85,B 0,C 180,E1 -27871.424,E2 -27871.424} C_VEL
LIN {X 0,Y 111.535,Z 210.487,A -85,B 0,C 180,E1 -27876.115,E2 -27876.115} C_VEL
LIN {X 0,Y 109.112,Z 206.736,A -85,B 0,C 180,E1 -27879.837,E2 -27879.837} C_VEL
LIN {X 0,Y 106.94,Z 203.284,A -85,B 0,C 180,E1 -27884.057,E2 -27884.057} C_VEL
LIN {X 0,Y 106.323,Z 202.482,A -85,B 0,C 180,E1 -27885.461,E2 -27885.461} C_VEL
LIN {X 0,Y 104.52,Z 199.931,A -85,B 0,C 180,E1 -27890.903,E2 -27890.903} C_VEL
LIN {X 0,Y 103.967,Z 197.965,A -85,B 0,C 180,E1 -27894.181,E2 -27894.181} C_VEL
LIN {X 0,Y 103.477,Z 197.362,A -85,B 0,C 180,E1 -27900,E2 -27900} C_VEL
LIN {X 0,Y 104.066,Z 198.246,A -85,B 0,C 180,E1 -27906.788,E2 -27906.788} C_VEL
LIN {X 0,Y 105.274,Z 201.381,A -85,B 0,C 180,E1 -27912.123,E2 -27912.123} C_VEL
LIN {X 0,Y 105.865,Z 203.07,A -85,B 0,C 180,E1 -27914.025,E2 -27914.025} C_VEL
LIN {X 0,Y 106.566,Z 207.735,A -85,B 0,C 180,E1 -27916.601,E2 -27916.601} C_VEL
LIN {X 0,Y 107.409,Z 212.694,A -85,B 0,C 180,E1 -27919.089,E2 -27919.089} C_VEL
LIN {X 0,Y 108.324,Z 214.818,A -85,B 0,C 180,E1 -27920.846,E2 -27920.846} C_VEL
LIN {X 0,Y 110.587,Z 218.822,A -85,B 0,C 180,E1 -27924.383,E2 -27924.383} C_VEL
LIN {X 0,Y 113.639,Z 224.63,A -85,B 0,C 180,E1 -27928.372,E2 -27928.372} C_VEL
LIN {X 0,Y 116.813,Z 231.447,A -85,B 0,C 180,E1 -27931.938,E2 -27931.938} C_VEL
LIN {X 0,Y 115.127,Z 243.651,A -85,B 0,C 180,E1 -27932.711,E2 -27932.711} C_VEL
LIN {X 0,Y 112.866,Z 253.428,A -85,B 0,C 180,E1 -27933.681,E2 -27933.681} C_VEL
LIN {X 0,Y 110.407,Z 261.416,A -85,B 0,C 180,E1 -27934.781,E2 -27934.781} C_VEL
LIN {X 0,Y 107.266,Z 269.578,A -85,B 0,C 180,E1 -27936.27,E2 -27936.27} C_VEL
LIN {X 0,Y 103.75,Z 277.105,A -85,B 0,C 180,E1 -27938.049,E2 -27938.049} C_VEL
LIN {X 0,Y 99.368,Z 285.007,A -85,B 0,C 180,E1 -27940.507,E2 -27940.507} C_VEL
LIN {X 0,Y 94.577,Z 292.377,A -85,B 0,C 180,E1 -27943.57,E2 -27943.57} C_VEL
LIN {X 0,Y 88.936,Z 299.845,A -85,B 0,C 180,E1 -27947.801,E2 -27947.801} C_VEL
LIN {X 0,Y 82.923,Z 306.683,A -85,B 0,C 180,E1 -27953.609,E2 -27953.609} C_VEL
LIN {X 0,Y 77.905,Z 311.853,A -85,B 0,C 180,E1 -27960.252,E2 -27960.252} C_VEL
LIN {X 0,Y 75.165,Z 314.502,A -85,B 0,C 180,E1 -27965.116,E2 -27965.116} C_VEL
LIN {X 0,Y 72.032,Z 317.402,A -85,B 0,C 180,E1 -27972.979,E2 -27972.979} C_VEL
LIN {X 0,Y 70.713,Z 318.662,A -85,B 0,C 180,E1 -27978.533,E2 -27978.533} C_VEL
LIN {X 0,Y 69.893,Z 319.455,A -85,B 0,C 180,E1 -27984.228,E2 -27984.228} C_VEL
LIN {X 0,Y 69.668,Z 319.756,A -85,B 0,C 180,E1 -27989.999,E2 -27989.999} C_VEL
LIN {X 0,Y 69.888,Z 319.474,A -85,B 0,C 180,E1 -27995.77,E2 -27995.77} C_VEL
LIN {X 0,Y 70.649,Z 318.72,A -85,B 0,C 180,E1 -28001.474,E2 -28001.474} C_VEL
LIN {X 0,Y 72.014,Z 317.498,A -85,B 0,C 180,E1 -28007.023,E2 -28007.023} C_VEL
LIN {X 0,Y 75.117,Z 314.638,A -85,B 0,C 180,E1 -28014.898,E2 -28014.898} C_VEL
LIN {X 0,Y 77.848,Z 312.032,A -85,B 0,C 180,E1 -28019.769,E2 -28019.769} C_VEL
LIN {X 0,Y 82.875,Z 306.91,A -85,B 0,C 180,E1 -28026.412,E2 -28026.412} C_VEL
LIN {X 0,Y 87.818,Z 301.396,A -85,B 0,C 180,E1 -28031.317,E2 -28031.317} C_VEL
LIN {X 0,Y 93.332,Z 294.46,A -85,B 0,C 180,E1 -28035.671,E2 -28035.671} C_VEL
LIN {X 0,Y 98.71,Z 286.495,A -85,B 0,C 180,E1 -28039.153,E2 -28039.153} C_VEL
LIN {X 0,Y 103.112,Z 278.901,A -85,B 0,C 180,E1 -28041.611,E2 -28041.611} C_VEL
LIN {X 0,Y 106.658,Z 271.658,A -85,B 0,C 180,E1 -28043.437,E2 -28043.437} C_VEL
LIN {X 0,Y 110.346,Z 262.493,A -85,B 0,C 180,E1 -28045.171,E2 -28045.171} C_VEL
LIN {X 0,Y 113.125,Z 253.55,A -85,B 0,C 180,E1 -28046.45,E2 -28046.45} C_VEL
LIN {X 0,Y 115.559,Z 242.932,A -85,B 0,C 180,E1 -28047.501,E2 -28047.501} C_VEL
LIN {X 0,Y 117.017,Z 231.614,A -85,B 0,C 180,E1 -28048.258,E2 -28048.258} C_VEL
LIN {X 0,Y 113.72,Z 224.553,A -85,B 0,C 180,E1 -28051.987,E2 -28051.987} C_VEL
LIN {X 0,Y 110.69,Z 218.793,A -85,B 0,C 180,E1 -28055.999,E2 -28055.999} C_VEL
LIN {X 0,Y 108.974,Z 215.79,A -85,B 0,C 180,E1 -28058.652,E2 -28058.652} C_VEL
LIN {X 0,Y 107.545,Z 213.305,A -85,B 0,C 180,E1 -28061.207,E2 -28061.207} C_VEL
LIN {X 0,Y 105.412,Z 209.569,A -85,B 0,C 180,E1 -28066.014,E2 -28066.014} C_VEL
LIN {X 0,Y 103.696,Z 207.056,A -85,B 0,C 180,E1 -28071.719,E2 -28071.719} C_VEL
LIN {X 0,Y 103.238,Z 205.125,A -85,B 0,C 180,E1 -28075.118,E2 -28075.118} C_VEL
LIN {X 0,Y 102.956,Z 204.653,A -85,B 0,C 180,E1 -28080.977,E2 -28080.977} C_VEL
LIN {X 0,Y 103.27,Z 205.299,A -85,B 0,C 180,E1 -28085.014,E2 -28085.014} C_VEL
LIN {X 0,Y 104.619,Z 208.756,A -85,B 0,C 180,E1 -28091.626,E2 -28091.626} C_VEL
LIN {X 0,Y 105.712,Z 210.097,A -85,B 0,C 180,E1 -28094.559,E2 -28094.559} C_VEL
LIN {X 0,Y 108.408,Z 214.737,A -85,B 0,C 180,E1 -28100.159,E2 -28100.159} C_VEL
LIN {X 0,Y 110.521,Z 218.468,A -85,B 0,C 180,E1 -28103.542,E2 -28103.542} C_VEL
LIN {X 0,Y 113.386,Z 223.844,A -85,B 0,C 180,E1 -28107.389,E2 -28107.389} C_VEL
LIN {X 0,Y 116.12,Z 229.728,A -85,B 0,C 180,E1 -28110.583,E2 -28110.583} C_VEL
LIN {X 0,Y 116.994,Z 232.714,A -85,B 0,C 180,E1 -28111.64,E2 -28111.64} C_VEL
LIN {X 0,Y 115.329,Z 245.344,A -85,B 0,C 180,E1 -28112.406,E2 -28112.406} C_VEL
LIN {X 0,Y 112.992,Z 255.129,A -85,B 0,C 180,E1 -28113.267,E2 -28113.267} C_VEL
LIN {X 0,Y 109.867,Z 264.859,A -85,B 0,C 180,E1 -28114.556,E2 -28114.556} C_VEL
LIN {X 0,Y 106.488,Z 273.133,A -85,B 0,C 180,E1 -28116.055,E2 -28116.055} C_VEL
LIN {X 0,Y 102.059,Z 282.147,A -85,B 0,C 180,E1 -28118.298,E2 -28118.298} C_VEL
LIN {X 0,Y 96.33,Z 291.651,A -85,B 0,C 180,E1 -28121.6,E2 -28121.6} C_VEL
LIN {X 0,Y 91.559,Z 298.244,A -85,B 0,C 180,E1 -28124.765,E2 -28124.765} C_VEL
LIN {X 0,Y 87.227,Z 303.734,A -85,B 0,C 180,E1 -28128.341,E2 -28128.341} C_VEL
LIN {X 0,Y 82.221,Z 309.28,A -85,B 0,C 180,E1 -28133.25,E2 -28133.25} C_VEL
LIN {X 0,Y 77.171,Z 314.44,A -85,B 0,C 180,E1 -28139.943,E2 -28139.943} C_VEL
LIN {X 0,Y 73.365,Z 318.23,A -85,B 0,C 180,E1 -28147.471,E2 -28147.471} C_VEL
LIN {X 0,Y 71.522,Z 319.968,A -85,B 0,C 180,E1 -28152.857,E2 -28152.857} C_VEL
LIN {X 0,Y 70.291,Z 321.212,A -85,B 0,C 180,E1 -28158.466,E2 -28158.466} C_VEL
LIN {X 0,Y 69.662,Z 321.983,A -85,B 0,C 180,E1 -28164.211,E2 -28164.211} C_VEL
LIN {X 0,Y 69.645,Z 322.276,A -85,B 0,C 180,E1 -28170.001,E2 -28170.001} C_VEL
LIN {X 0,Y 69.662,Z 321.969,A -85,B 0,C 180,E1 -28175.792,E2 -28175.792} C_VEL
LIN {X 0,Y 70.287,Z 321.169,A -85,B 0,C 180,E1 -28181.537,E2 -28181.537} C_VEL
LIN {X 0,Y 71.506,Z 319.897,A -85,B 0,C 180,E1 -28187.15,E2 -28187.15} C_VEL
LIN {X 0,Y 74.472,Z 316.972,A -85,B 0,C 180,E1 -28195.131,E2 -28195.131} C_VEL
LIN {X 0,Y 77.162,Z 314.308,A -85,B 0,C 180,E1 -28200.064,E2 -28200.064} C_VEL
LIN {X 0,Y 82.196,Z 309.11,A -85,B 0,C 180,E1 -28206.765,E2 -28206.765} C_VEL
LIN {X 0,Y 88.284,Z 302.254,A -85,B 0,C 180,E1 -28212.584,E2 -28212.584} C_VEL
LIN {X 0,Y 93.908,Z 294.767,A -85,B 0,C 180,E1 -28216.861,E2 -28216.861} C_VEL
LIN {X 0,Y 98.772,Z 287.384,A -85,B 0,C 180,E1 -28219.9,E2 -28219.9} C_VEL
LIN {X 0,Y 103.027,Z 279.842,A -85,B 0,C 180,E1 -28222.228,E2 -28222.228} C_VEL
LIN {X 0,Y 107.173,Z 271.105,A -85,B 0,C 180,E1 -28224.245,E2 -28224.245} C_VEL
LIN {X 0,Y 111.091,Z 260.782,A -85,B 0,C 180,E1 -28225.978,E2 -28225.978} C_VEL
LIN {X 0,Y 114.305,Z 248.945,A -85,B 0,C 180,E1 -28227.228,E2 -28227.228} C_VEL
LIN {X 0,Y 115.987,Z 239.395,A -85,B 0,C 180,E1 -28227.912,E2 -28227.912} C_VEL
LIN {X 0,Y 116.731,Z 232.432,A -85,B 0,C 180,E1 -28228.315,E2 -28228.315} C_VEL
LIN {X 0,Y 115.436,Z 228.398,A -85,B 0,C 180,E1 -28229.849,E2 -28229.849} C_VEL
LIN {X 0,Y 112.212,Z 221.862,A -85,B 0,C 180,E1 -28233.703,E2 -28233.703} C_VEL
LIN {X 0,Y 109.26,Z 216.394,A -85,B 0,C 180,E1 -28237.921,E2 -28237.921} C_VEL
LIN {X 0,Y 107.396,Z 213.227,A -85,B 0,C 180,E1 -28241.124,E2 -28241.124} C_VEL
LIN {X 0,Y 105.149,Z 209.389,A -85,B 0,C 180,E1 -28246.093,E2 -28246.093} C_VEL
LIN {X 0,Y 103.453,Z 206.833,A -85,B 0,C 180,E1 -28251.639,E2 -28251.639} C_VEL
LIN {X 0,Y 102.95,Z 204.903,A -85,B 0,C 180,E1 -28255.105,E2 -28255.105} C_VEL
LIN {X 0,Y 102.613,Z 204.4,A -85,B 0,C 180,E1 -28260,E2 -28260} C_VEL
LIN {X 0,Y 103.069,Z 205.233,A -85,B 0,C 180,E1 -28266.116,E2 -28266.116} C_VEL
LIN {X 0,Y 104.141,Z 208.268,A -85,B 0,C 180,E1 -28271.405,E2 -28271.405} C_VEL
LIN {X 0,Y 105.479,Z 209.907,A -85,B 0,C 180,E1 -28275.04,E2 -28275.04} C_VEL
LIN {X 0,Y 107.734,Z 213.691,A -85,B 0,C 180,E1 -28279.78,E2 -28279.78} C_VEL
LIN {X 0,Y 108.324,Z 214.818,A -85,B 0,C 180,E1 -28280.846,E2 -28280.846} C_VEL
LIN {X 0,Y 109.242,Z 217.019,A -85,B 0,C 180,E1 -28282.461,E2 -28282.461} C_VEL
LIN {X 0,Y 109.831,Z 220.15,A -85,B 0,C 180,E1 -28283.705,E2 -28283.705} C_VEL
LIN {X 0,Y 111.066,Z 229.638,A -85,B 0,C 180,E1 -28286.514,E2 -28286.514} C_VEL
LIN {X 0,Y 111.679,Z 231.652,A -85,B 0,C 180,E1 -28287.42,E2 -28287.42} C_VEL
LIN {X 0,Y 112.87,Z 234.507,A -85,B 0,C 180,E1 -28289.026,E2 -28289.026} C_VEL
LIN {X 0,Y 111.334,Z 244.38,A -85,B 0,C 180,E1 -28289.696,E2 -28289.696} C_VEL
LIN {X 0,Y 109.258,Z 253.022,A -85,B 0,C 180,E1 -28290.524,E2 -28290.524} C_VEL
LIN {X 0,Y 106.464,Z 261.706,A -85,B 0,C 180,E1 -28291.672,E2 -28291.672} C_VEL
LIN {X 0,Y 103.23,Z 269.711,A -85,B 0,C 180,E1 -28293.096,E2 -28293.096} C_VEL
LIN {X 0,Y 99.546,Z 277.237,A -85,B 0,C 180,E1 -28294.84,E2 -28294.84} C_VEL
LIN {X 0,Y 94.917,Z 285.138,A -85,B 0,C 180,E1 -28297.252,E2 -28297.252} C_VEL
LIN {X 0,Y 89.843,Z 292.508,A -85,B 0,C 180,E1 -28300.296,E2 -28300.296} C_VEL
LIN {X 0,Y 83.822,Z 299.976,A -85,B 0,C 180,E1 -28304.545,E2 -28304.545} C_VEL
LIN {X 0,Y 77.32,Z 306.813,A -85,B 0,C 180,E1 -28310.485,E2 -28310.485} C_VEL
LIN {X 0,Y 71.824,Z 311.983,A -85,B 0,C 180,E1 -28317.439,E2 -28317.439} C_VEL
LIN {X 0,Y 68.775,Z 314.631,A -85,B 0,C 180,E1 -28322.621,E2 -28322.621} C_VEL
LIN {X 0,Y 65.272,Z 317.531,A -85,B 0,C 180,E1 -28331.153,E2 -28331.153} C_VEL
LIN {X 0,Y 63.766,Z 318.791,A -85,B 0,C 180,E1 -28337.264,E2 -28337.264} C_VEL
LIN {X 0,Y 62.835,Z 319.583,A -85,B 0,C 180,E1 -28343.577,E2 -28343.577} C_VEL
LIN {X 0,Y 62.569,Z 319.884,A -85,B 0,C 180,E1 -28349.998,E2 -28349.998} C_VEL
LIN {X 0,Y 62.829,Z 319.602,A -85,B 0,C 180,E1 -28356.421,E2 -28356.421} C_VEL
LIN {X 0,Y 63.715,Z 318.848,A -85,B 0,C 180,E1 -28362.743,E2 -28362.743} C_VEL
LIN {X 0,Y 65.256,Z 317.626,A -85,B 0,C 180,E1 -28368.849,E2 -28368.849} C_VEL
LIN {X 0,Y 68.73,Z 314.766,A -85,B 0,C 180,E1 -28377.395,E2 -28377.395} C_VEL
LIN {X 0,Y 71.775,Z 312.159,A -85,B 0,C 180,E1 -28382.583,E2 -28382.583} C_VEL
LIN {X 0,Y 77.27,Z 307.037,A -85,B 0,C 180,E1 -28389.542,E2 -28389.542} C_VEL
LIN {X 0,Y 82.62,Z 301.523,A -85,B 0,C 180,E1 -28394.568,E2 -28394.568} C_VEL
LIN {X 0,Y 88.525,Z 294.585,A -85,B 0,C 180,E1 -28398.954,E2 -28398.954} C_VEL
LIN {X 0,Y 94.22,Z 286.621,A -85,B 0,C 180,E1 -28402.421,E2 -28402.421} C_VEL
LIN {X 0,Y 98.858,Z 279.025,A -85,B 0,C 180,E1 -28404.839,E2 -28404.839} C_VEL
LIN {X 0,Y 102.771,Z 271.388,A -85,B 0,C 180,E1 -28406.701,E2 -28406.701} C_VEL
LIN {X 0,Y 106.454,Z 262.612,A -85,B 0,C 180,E1 -28408.309,E2 -28408.309} C_VEL
LIN {X 0,Y 109.039,Z 254.817,A -85,B 0,C 180,E1 -28409.408,E2 -28409.408} C_VEL
LIN {X 0,Y 111.438,Z 245.292,A -85,B 0,C 180,E1 -28410.374,E2 -28410.374} C_VEL
LIN {X 0,Y 113.071,Z 235.358,A -85,B 0,C 180,E1 -28411.055,E2 -28411.055} C_VEL
LIN {X 0,Y 112.961,Z 234.296,A -85,B 0,C 180,E1 -28411.348,E2 -28411.348} C_VEL
LIN {X 0,Y 109.903,Z 227.521,A -85,B 0,C 180,E1 -28415.549,E2 -28415.549} C_VEL
LIN {X 0,Y 107.387,Z 222.522,A -85,B 0,C 180,E1 -28419.636,E2 -28419.636} C_VEL
LIN {X 0,Y 105.881,Z 219.715,A -85,B 0,C 180,E1 -28422.589,E2 -28422.589} C_VEL
LIN {X 0,Y 104.013,Z 216.231,A -85,B 0,C 180,E1 -28427.314,E2 -28427.314} C_VEL
LIN {X 0,Y 102.538,Z 213.541,A -85,B 0,C 180,E1 -28433.234,E2 -28433.234} C_VEL
LIN {X 0,Y 102.263,Z 212.008,A -85,B 0,C 180,E1 -28436.059,E2 -28436.059} C_VEL
LIN {X 0,Y 102.091,Z 211.695,A -85,B 0,C 180,E1 -28440.986,E2 -28440.986} C_VEL
LIN {X 0,Y 102.298,Z 212.232,A -85,B 0,C 180,E1 -28444.22,E2 -28444.22} C_VEL
LIN {X 0,Y 103.524,Z 215.682,A -85,B 0,C 180,E1 -28451.007,E2 -28451.007} C_VEL
LIN {X 0,Y 104.367,Z 216.886,A -85,B 0,C 180,E1 -28453.508,E2 -28453.508} C_VEL
LIN {X 0,Y 106.644,Z 221.114,A -85,B 0,C 180,E1 -28458.759,E2 -28458.759} C_VEL
LIN {X 0,Y 108.595,Z 224.875,A -85,B 0,C 180,E1 -28462.221,E2 -28462.221} C_VEL
LIN {X 0,Y 111.556,Z 230.979,A -85,B 0,C 180,E1 -28466.545,E2 -28466.545} C_VEL
LIN {X 0,Y 113.103,Z 234.845,A -85,B 0,C 180,E1 -28468.582,E2 -28468.582} C_VEL
LIN {X 0,Y 112.806,Z 238.186,A -85,B 0,C 180,E1 -28468.897,E2 -28468.897} C_VEL
LIN {X 0,Y 111.226,Z 247.165,A -85,B 0,C 180,E1 -28469.447,E2 -28469.447} C_VEL
LIN {X 0,Y 108.893,Z 256.217,A -85,B 0,C 180,E1 -28470.281,E2 -28470.281} C_VEL
